(* IEC 61131-3 sources: Mizera_Tube/Plc (part 3) *)

(* ---- LASER.plc ---- *)
*******************************************************************************
*   LASER.PLC
*   ESAutomotion
*   LASER machine
*******************************************************************************
#funcdec "FLP.plc"
#funcdec "RestFB.plc"
VAR
#include "Cnc.inc"

#include "RemContr.inc"

HoerbEnabCond: BOOL; * Hoerbiger prop. valve enable conditions
TOF_HBPROP: TOF;
#defcom TOF_HBPROP.Q Hoerbiger prop valve enable delayed

appoggio:             BOOL;

TP_HOLD_Tip:                TP;
TP_HOLD_Noz:                TP;

F_DIS_MANAPA:               F_TRIG;

R_TRIG_PRGRUN:              R_TRIG; * Fronte salita start programma
R_TRIG_PRGRUN2:             R_TRIG; * Fronte salita start programma
F_TRIG_PRGRUN:              F_TRIG; * Fronte discesa start programma

R_TRIG0:                    R_TRIG;
TON_ST:                        TON;

*manual cut
TP_EXE_REQ:                 TP;
FTRIG_PRUN:                 F_TRIG;
TP_EXE_REQ2:                TP;
FTRIG_PRUN2:                F_TRIG;
RTRIG_Xstart:               R_TRIG;
RTRIG_Xend:                 R_TRIG;
RTRIG_Ystart:               R_TRIG;
RTRIG_Yend:                 R_TRIG;
RTRIG_REQ_BREAK:            R_TRIG;
*
* microjoint alg
firScan:                   DWORD;                * Initialization of filter
RTRIG_FIR_INIT:           R_TRIG;
error:                     DWORD;
TON_VALID_DATA:              TON;

TON_DISABLE_BEAM:            TON;
RTRIG_CAL_FILTER:         R_TRIG;
velMaxAlg:                 DWORD;                 * set point speed to have filter at 0
RTRIG_START_LEAD:         R_TRIG;
FTRIG_START_LEAD:         F_TRIG;
posXinitlead:              DWORD;
posYinitlead:              DWORD;
posXendlead:               DWORD;
posYendlead:               DWORD;
PosIntInitLead:            DWORD;
PosIntendLead:             DWORD;
microJoinfactor:           DWORD;        * need to comensate the possible radius during lead in
percReduction:             DWORD;
LinearDistance:            DWORD;
RealLeadDistance:          DWORD;
distX:                     DWORD;
distY:                     DWORD;
indexLeadIn:               DWORD;        * if  indexLeadIn = 314 lead in is a semicircumference
Ftrig_LeadTest:           F_TRIG;

RTRIG_COUNT_PIERC:        R_TRIG;
rtrig_ResPiercCounter:    R_TRIG;
rtrig_ResPiercCounter_2:  R_TRIG;
MicroJointime:         DWORD;

* wrong operation protection

RTRIG_NOPIERC:            R_TRIG;
RTRIG_ALLPIERC:           R_TRIG;
RTRIG_NOLEAD:             R_TRIG;
RTRIG_RES_GEOM:           R_TRIG;
RTRIG_RES_PIECE:          R_TRIG;
FTRIG_RES_AUTO_CLEAN:     F_TRIG;
RTRIG_WORK_ENAB:          R_TRIG;

TP_BUZZER:              TP;         * Buzzer timer
TP_HOLD_BODY:           TP;

TON_REMOVE_ALARM:       TON;
RTRIG_ORIG19:           R_TRIG;
RTRIG_BLOCK_S:          R_TRIG;

RTRIG_MANSEL_P:         R_TRIG;         * Selettore manuale (potenza/duty/frequenza)
RTRIG_MANSEL_M:         R_TRIG;         * Selettore manuale (potenza/duty/frequenza)

Restart:                Restart_Cut;

END_VAR

VAR_IN_OUT
#include "mem.inc"
END_VAR

#include "Iol.inc"

******************************************************************************
* FUNCTION LASER_IN
******************************************************************************
FUNCTION LASER_IN

**@@@ INP_TEST    * Digital Inputs test management

******************************************************************************
*   Gestione selettore manuale x cambiamento valori potenza/duty/frequenza
******************************************************************************
CAL  RTRIG_MANSEL_P (CLK:=%SoftBtn1.0)
CAL  RTRIG_MANSEL_M (CLK:=%SoftBtn1.1)

*** INC

LD   ON_ONE_SCAN                   ** PLCFLAGS.8  Flag on alla prima scansione PLC
OR (
LD   ManSelector            *(rgGui6)Selettore manuale potenza/duty/frequenza
LE   0
)
OR (
LD   ManSelector            *(rgGui6)Selettore manuale potenza/duty/frequenza
GT   3
)
JMPCN man_sel_init

LD   100
ST   ManSelectorPOW         *(rgGui7)Selettore manuale POTENZA: ultimo valore impostato
ST   ManSelectorDUTY        *(rgGui8)Selettore manuale DUTY: ultimo valore impostato
ST   ManSelectorFREQ        *(rgGui9)Selettore manuale FREQUENCY: ultimo valore impostato

man_sel_init:

LD   RTRIG_MANSEL_P.Q
AND (
LD   ManSelector            *(rgGui6)Selettore manuale potenza/duty/frequenza
EQ   1
)
JMPCN no_pow_inc

LD   ManSelectorPOW         *(rgGui7)Selettore manuale POTENZA: ultimo valore impostato
ADD  1
ST   ManSelectorPOW         *(rgGui7)Selettore manuale POTENZA: ultimo valore impostato

no_pow_inc:
LD   RTRIG_MANSEL_P.Q
AND (
LD   ManSelector            *(rgGui6)Selettore manuale potenza/duty/frequenza
EQ   2
)
JMPCN no_duty_inc

LD   ManSelectorDUTY        *(rgGui8)Selettore manuale DUTY: ultimo valore impostato
ADD  5
ST   ManSelectorDUTY        *(rgGui8)Selettore manuale DUTY: ultimo valore impostato

no_duty_inc:
LD   RTRIG_MANSEL_P.Q
AND (
LD   ManSelector            *(rgGui6)Selettore manuale potenza/duty/frequenza
EQ   3
)
JMPCN no_freq_inc

LD   ManSelectorFREQ        *(rgGui9)Selettore manuale FREQUENCY: ultimo valore impostato
ADD  5
ST   ManSelectorFREQ        *(rgGui9)Selettore manuale FREQUENCY: ultimo valore impostato

no_freq_inc:

*** DEC

LD   RTRIG_MANSEL_M.Q
AND (
LD   ManSelector            *(rgGui6)Selettore manuale potenza/duty/frequenza
EQ   1
)
JMPCN no_pow_dec

LD   ManSelectorPOW         *(rgGui7)Selettore manuale POTENZA: ultimo valore impostato
SUB  1
ST   ManSelectorPOW         *(rgGui7)Selettore manuale POTENZA: ultimo valore impostato

no_pow_dec:
LD   RTRIG_MANSEL_M.Q
AND (
LD   ManSelector            *(rgGui6)Selettore manuale potenza/duty/frequenza
EQ   2
)
JMPCN no_duty_dec

LD   ManSelectorDUTY        *(rgGui8)Selettore manuale DUTY: ultimo valore impostato
SUB  5
ST   ManSelectorDUTY        *(rgGui8)Selettore manuale DUTY: ultimo valore impostato

no_duty_dec:
LD   RTRIG_MANSEL_M.Q
AND (
LD   ManSelector            *(rgGui6)Selettore manuale potenza/duty/frequenza
EQ   3
)
JMPCN no_freq_dec

LD   ManSelectorFREQ        *(rgGui9)Selettore manuale FREQUENCY: ultimo valore impostato
SUB  5
ST   ManSelectorFREQ        *(rgGui9)Selettore manuale FREQUENCY: ultimo valore impostato

no_freq_dec:

*** CONTROLLO VALORE MINIMO/MASSIMO

LD   ManSelectorPOW         *(rgGui7)Selettore manuale POTENZA: ultimo valore impostato
LT   0
JMPCN no_pow_zero
LD   0
ST   ManSelectorPOW         *(rgGui7)Selettore manuale POTENZA: ultimo valore impostato
no_pow_zero:
LD   ManSelectorPOW         *(rgGui7)Selettore manuale POTENZA: ultimo valore impostato
GT   120
JMPCN no_pow_max
LD   120
ST   ManSelectorPOW         *(rgGui7)Selettore manuale POTENZA: ultimo valore impostato
no_pow_max:

LD   ManSelectorDUTY        *(rgGui8)Selettore manuale DUTY: ultimo valore impostato
LT   0
JMPCN no_duty_zero
LD   0
ST   ManSelectorDUTY        *(rgGui8)Selettore manuale DUTY: ultimo valore impostato
no_duty_zero:
LD   ManSelectorDUTY        *(rgGui8)Selettore manuale DUTY: ultimo valore impostato
GT   120
JMPCN no_duty_max
LD   120
ST   ManSelectorDUTY        *(rgGui8)Selettore manuale DUTY: ultimo valore impostato
no_duty_max:

LD   ManSelectorFREQ        *(rgGui9)Selettore manuale FREQUENCY: ultimo valore impostato
LT   0
JMPCN no_freq_zero
LD   0
ST   ManSelectorFREQ        *(rgGui9)Selettore manuale FREQUENCY: ultimo valore impostato
no_freq_zero:
LD   ManSelectorFREQ        *(rgGui9)Selettore manuale FREQUENCY: ultimo valore impostato
GT   120
JMPCN no_freq_max
LD   120
ST   ManSelectorFREQ        *(rgGui9)Selettore manuale FREQUENCY: ultimo valore impostato
no_freq_max:

*** VALORI DI USCITA PER LsrGest.plc

LD   0
ST   ManSelectorPOW_out         *(gPlc30)Selettore manuale POTENZA: ultimo valore impostato (valore di uscita per LsrGest)
ST   ManSelectorDUTY_out        *(gPlc30)Selettore manuale DUTY: ultimo valore impostato (valore di uscita per LsrGest)
ST   ManSelectorFREQ_out        *(gPlc30)Selettore manuale FREQUENCY: ultimo valore impostato (valore di uscita per LsrGest)

LD   ManSelector            *(rgGui6)Selettore manuale potenza/duty/frequenza
EQ   1
JMPCN no_pow

LD   100
ST   ManSelectorDUTY        *(rgGui8)Selettore manuale DUTY: ultimo valore impostato
ST   ManSelectorFREQ        *(rgGui9)Selettore manuale FREQUENCY: ultimo valore impostato
JMP  no_freq

no_pow:
LD   ManSelector            *(rgGui6)Selettore manuale potenza/duty/frequenza
EQ   2
JMPCN no_duty

LD   100
ST   ManSelectorPOW         *(rgGui7)Selettore manuale POTENZA: ultimo valore impostato
ST   ManSelectorFREQ        *(rgGui9)Selettore manuale FREQUENCY: ultimo valore impostato
JMP  no_freq

no_duty:
LD   ManSelector            *(rgGui6)Selettore manuale potenza/duty/frequenza
EQ   3
JMPCN no_freq

LD   100
ST   ManSelectorPOW         *(rgGui7)Selettore manuale POTENZA: ultimo valore impostato
ST   ManSelectorDUTY        *(rgGui8)Selettore manuale DUTY: ultimo valore impostato

LD   %TabLsr0.L_CutFreq
MUL (
LD   ManSelectorFREQ        *(rgGui9)Selettore manuale FREQUENCY: ultimo valore impostato
SUB  100                    * 100%
)
DIV  100                    * 100 %
ST   ManSelectorFREQ_out        *(gPlc30)Selettore manuale FREQUENCY: ultimo valore impostato (valore di uscita per LsrGest)

no_freq:

******************************************************************************
*   Copia il valore della potenza massima sulla variabile usata dalla GUI
******************************************************************************
LD   %LsrGest0.ParMaxPower
ST   PotenzaMaxLaser            **(rLsGui17)Potenza massima Laser

******************************************************************************
* Safety for axes when operator move in jog the axes
CAL  TON_REMOVE_ALARM (IN:=%PLCerr7.21,PT:=5000)    * Axes cannot move, not safe movement

LD   OrderMoveYPosit               ** (LsPlc26.5) Order of movement positive dir for Y
OR   OrderMoveYNegat               ** (LsPlc26.6) Order of movement negative dir for Y
OR   OrderMoveXPosit               ** (LsPlc26.3) Order of movement positive dir for X
OR   OrderMoveXNegat               ** (LsPlc26.4) Order of movement negative dir for X
OR   Pul_Reset                     ** (gPlc0.3)Reset pushbutton
OR   TON_REMOVE_ALARM.Q        * Reset of the alarm
OR   PRGRUN_CN0                    ** M0.0 cn0.rc8.0  Programma in corso
R    %PLCerr7.21               * Axes cannot move, not safe movement

LD   %CalPipe0.General0.5       * pipe is along Y axis
AND  %cn3.cc1.5                 * W axis configured
ANDN PRGRUN_CN0                    ** M0.0 cn0.rc8.0  Programma in corso
ANDN BCI_TAR                       ** rc0.8  Selettore modi operativi su REF (taratura)
JMPCN noPipeY

  * hold moving if the bridge in in the middle of the machine and
  * the operator move X in pipe side
  LD   %ax28.ra4                  * y axis position
  SUB  3000
  GT   %tab1.t_ttab.t_oart.t_dY   * pipe offset along y axis
  OR  (
  LD   %ax29.ra4
  LE  (
  LD   %ax29.pa22
  SUB  10000
  )
  )
  AND  (
  LD   %ax27.ra4                  * x axis position
  LE   (
  LD   %ax27.pa21
  ADD  SafePipeZone                  ** (%LSRCostK9) Safety distance from axis limit in pipe management
   )
  )
  AND  (
  LD  %tab1.t_ttab.t_oart.t_dX
  LT  0
  )
  AND OrderMoveXNegat                ** (LsPlc26.4) Order of movement negative dir for X
 ***************************
  OR  ( * x is in the pipe side but head is not up
  LD   %ax27.ra4                  * x axis position
  LT   (
  LD   %ax27.pa21
  ADD  SafePipeZone                  ** (%LSRCostK9) Safety distance from axis limit in pipe management
   )
  AND (
  LD   %ax29.ra4
  LE  (
  LD   %ax29.pa22
  SUB  10000
    )
   )
  AND  OrderMoveXPosit               ** (LsPlc26.3) Order of movement positive dir for X
  ANDN (
  LD   %ax28.ra4                  * y axis position
  SUB  3000
  GT   %tab1.t_ttab.t_oart.t_dY   * pipe offset along y axis
  )
  AND  (
  LD  %tab1.t_ttab.t_oart.t_dX
  LT  0
  )
  )
 **************************
  OR  (  * same condition, in case the pipe is in positive direction of X axis
   LD   %ax28.ra4                  * y axis position
   SUB  3000
   GT   %tab1.t_ttab.t_oart.t_dY   * pipe offset along y axis
   OR  (
   LD   %ax29.ra4
   LE  (
   LD   %ax29.pa22
   SUB  10000
    )
   )
   AND  (
   LD   %ax27.ra4                  * x axis position
   GE   (
   LD   %ax27.pa22
   SUB  SafePipeZone                  ** (%LSRCostK9) Safety distance from axis limit in pipe management
    )
   )
   AND  (
   LD  %tab1.t_ttab.t_oart.t_dX
   GT  0
   )
   AND  OrderMoveXPosit               ** (LsPlc26.3) Order of movement positive dir for X
  )
 ***************************
  OR  ( * x is in the pipe side but head is not up
  LD   %ax27.ra4                  * x axis position
  GE   (
  LD   %ax27.pa22
  SUB  SafePipeZone                  ** (%LSRCostK9) Safety distance from axis limit in pipe management
   )
  AND (
  LD   %ax29.ra4
  LE  (
  LD   %ax29.pa22
  SUB  10000
    )
   )
  AND  OrderMoveXNegat               ** (LsPlc26.4) Order of movement negative dir for X
  ANDN (
  LD   %ax28.ra4                  * y axis position
  SUB  3000
  GT   %tab1.t_ttab.t_oart.t_dY   * pipe offset along y axis
  )
  AND  (
  LD  %tab1.t_ttab.t_oart.t_dX
  GT  0
   )
  )
 **************************
  ST  HoldSafePipeX                  ** (LsPlc26.2) Hold moving for X axis, not allow manual movement in pipe area

  LD   %ax27.ra4                  * x axis position
  LT   (
  LD   %ax27.pa21
  ADD  SafePipeZone                  ** (%LSRCostK9) Safety distance from axis limit in pipe management
   )
  AND  (
  LD  %tab1.t_ttab.t_oart.t_dX
  LT  0
  )
  AND (
  LD  OrderMoveYPosit                ** (LsPlc26.5) Order of movement positive dir for Y
  OR  OrderMoveYNegat                ** (LsPlc26.6) Order of movement negative dir for Y
  )
  OR  (
   LD   %ax27.ra4                 * x axis position
   GT   (
   LD   %ax27.pa22
   SUB  SafePipeZone                  ** (%LSRCostK9) Safety distance from axis limit in pipe management
    )
    AND  (
    LD  %tab1.t_ttab.t_oart.t_dX
    GT  0
   )
    AND (
    LD  OrderMoveYPosit                ** (LsPlc26.5) Order of movement positive dir for Y
    OR  OrderMoveYNegat                ** (LsPlc26.6) Order of movement negative dir for Y
   )
  )
  ST   HoldSafePipeY                 ** (LsPlc26.7) Hold moving for Y axis, not allow manual movement in pipe area

noPipeY:

* Safety for axes when operator move in jog the axes
* NEED TO BE TESTED,ACTUALLY MACHINE HAVE PIPE ALONG y

LD   %CalPipe0.General0.4       * pipe is along X axis
AND  %cn3.cc1.5                 * W axis configured
ANDN PRGRUN_CN0                    ** M0.0 cn0.rc8.0  Programma in corso
ANDN BCI_TAR                       ** rc0.8  Selettore modi operativi su REF (taratura)
JMPCN noPipeX

  LD   %ax27.ra4                  * x axis position
  SUB  3000
  GT   %tab1.t_ttab.t_oart.t_dX   * pipe offset along x axis
  AND  (
  LD   %ax28.ra4                  * y axis position
  LT   (
  LD   %ax28.pa21
  ADD  SafePipeZone                  ** (%LSRCostK9) Safety distance from axis limit in pipe management
   )
  )
  AND  (
  LD  %tab1.t_ttab.t_oart.t_dY
  LT  0
  )
  AND OrderMoveYNegat                ** (LsPlc26.6) Order of movement negative dir for Y
  OR  (
   LD   %ax27.ra4                  * x axis position
   SUB  3000
   GT   %tab1.t_ttab.t_oart.t_dX   * pipe offset along y axis
   AND  (
   LD   %ax28.ra4                  * y axis position
   GT   (
   LD   %ax28.pa22
   SUB  SafePipeZone                  ** (%LSRCostK9) Safety distance from axis limit in pipe management
    )
   )
   AND  (
   LD  %tab1.t_ttab.t_oart.t_dY
   GT  0
   )
   AND  OrderMoveYPosit               ** (LsPlc26.5) Order of movement positive dir for Y
  )
  ST  HoldSafePipeY                  ** (LsPlc26.7) Hold moving for Y axis, not allow manual movement in pipe area

  LD   %ax28.ra4                   * y axis position
  LT   (
  LD   %ax28.pa21
  ADD  SafePipeZone                  ** (%LSRCostK9) Safety distance from axis limit in pipe management
   )
  AND  (
  LD  %tab1.t_ttab.t_oart.t_dY
  LT  0
  )
  AND (
  LD  OrderMoveYPosit                ** (LsPlc26.5) Order of movement positive dir for Y
  OR  OrderMoveYNegat                ** (LsPlc26.6) Order of movement negative dir for Y
  )
  OR  (
   LD   %ax28.ra4                  * y axis position
   GT   (
   LD   %ax28.pa22
   SUB  SafePipeZone                  ** (%LSRCostK9) Safety distance from axis limit in pipe management
    )
    AND  (
    LD  %tab1.t_ttab.t_oart.t_dY
    GT  0
   )
    AND (
    LD  OrderMoveYPosit                ** (LsPlc26.5) Order of movement positive dir for Y
    OR  OrderMoveYNegat                ** (LsPlc26.6) Order of movement negative dir for Y
   )
  )
  ST   HoldSafePipeX                 ** (LsPlc26.2) Hold moving for X axis, not allow manual movement in pipe area

noPipeX:

LD   HoldSafePipeX                 ** (LsPlc26.2) Hold moving for X axis, not allow manual movement in pipe area
OR   HoldSafePipeY                 ** (LsPlc26.7) Hold moving for Y axis, not allow manual movement in pipe area
S    %PLCerr7.21                    * Axes cannot move, not safe movement

******************************************************************************
******************************************************************************
*   BUZZER MANAGEMENT
******************************************************************************
LD   PRGRUN_CN0                    ** M0.0 cn0.rc8.0  Programma in corso
ST   appoggio

CAL  TP_BUZZER(IN=PRGRUN_CN0,PT=%Cost_User20) ** Buzzer timer

LD   TP_BUZZER.Q
ST	 O_O_BUZZER_START_CIC           ** Star cycle buzzer

******************************************************************************
CAL  TP_HOLD_Tip(IN=%PLCerr5.4,PT=500) **PLC Err 164 Tip touch (A11=1, A14=0, A15=0 in normal operation)
CAL  TP_HOLD_Noz(IN=%PLCerr5.6,PT=1000) **PLC Err 166 Nozzle lost (A11=1, A14=0, A15=1 in normal operation)
CAL  TP_HOLD_BODY (IN:=%PLCerr5.5,PT:=1000)                    **PLC Err 165 Body touch (A11=1, A14=1, A15=0 in normal operation)

LD   TP_HOLD_Tip.Q
OR   TP_HOLD_Noz.Q
OR   TP_HOLD_BODY.Q
ST   StopUsrPlc                    ** (gPlc2.22)Richiesta STOP da User_Plc

**************************************
*& Set TAB value for startup (retentive)
**
LD      ON_ONE_SCAN                ** PLCFLAGS.8  Flag on alla prima scansione PLC
JMPCN   No_FirstScan
  LD      guiTAB_Sinottico           ** (rGui10)GUI TAB Sinottico for Quotes
  EQ      0
  JMPCN   No_TabEqZero
    LD      1
    ST      guiTAB_Sinottico           ** (rGui10)GUI TAB Sinottico for Quotes
No_TabEqZero:
No_FirstScan:

CAL R_TRIG0(CLK=%PLCFLAGS.10)

LD   R_TRIG0.Q
JMPCN CNT_MP

LD   Timesec                       ** (R123) Tempo secondi
ADD  1
ST   Timesec                       ** (R123) Tempo secondi

CNT_MP:

LD   Timesec                       ** (R123) Tempo secondi
DIV  3600
ST   TimeOur                       ** (R124) Tempo ore
****************************************************************

****************************************************************
* Tempo Taglio In Corso
****************************************************************

CAL  TON_ST(IN:=StartTimer,PT:=1000) ** Start tim

LD   %cn0.rc8.0                    * Programma in corso cn0
AND  TON_ST.Q                     * Start tim
ANDN PRGSTOP_CN0                   ** (cn0.rc8.1)  Programma interrotto CN0
AND  R_TRIG0.Q                     * Impulso incremento secondi
JMPCN TIMECUT

* Contasecondi

LD   TimeSecProg                   ** (R125) Conteggio Secondi Tempo Programma Taglio in corso
ADD  1
ST   TimeSecProg                   ** (R125) Conteggio Secondi Tempo Programma Taglio in corso

TIMECUT:

CAL R_TRIG_PRGRUN(CLK=%cn0.rc8.0)	 ** Fronte salita start programma

LD   R_TRIG_PRGRUN.Q
JMPCN ResCount

LD   0
ST   TimeSecProg                   ** (R125) Conteggio Secondi Tempo Programma Taglio in corso
ST   TimeMinProg                   ** (R126) Conteggio Minuti Tempo Programma Taglio in corso

ResCount:

LD   Pul_Reset                     ** (gPlc0.3)Reset pushbutton
JMPCN no_zero
LD   0
ST   StartTimer                    ** Start tim
no_zero:

*******************************************************************************
*   Restart Taglio
*******************************************************************************
LD   PRGRUN_CN0
ST   Restart.xProg_Run

LD   %PLCerr5.4                    **PLC Err 164 Tip touch (A11=1, A14=0, A15=0 in normal operation)
AND  EnTiptouchRetrace
AND  BevelHeadSyncG800              * Traccia in esecuzione
ST   Restart.xTip_Touch

LD   VRTCIncSetPReached
ST   Restart.xZupExecuted

LD   PRGSTOP_CN0
ST   Restart.xMachineInHold

LD   %LSRCostK13                    ** (LSRCostK13) Numero tentativi per tip touch con gestione autorestart
ST   Restart.xAttempts

LD   RetraceCommBack
ST   Restart.xRetraceOn

CAL  Restart

LD   Restart.yStartProg
ST   StartAftTipTouch              ** (LsPlc47.2) Start after tip touch

LD   Restart.yStartRetrace
ST   JogCommandTipTouch            ** (LsPlc47.0) Automatic jog command for tip touch

LD   Restart.yZupRequest
ST   EnPosiz                       * (LsPlc47.3) Abilitaz. posiz. Asse Z

LD   Restart.yInibTipTouch
AND  EnTiptouchRetrace
ST   InibTipTouchAllarm            ** M100.22 Inibizione allarme Tip Touch per restart ciclo

**********************************************************************************
* enable/disable automatic height control manual cut

LD   %cn0.rc9            * Channel 0 M-Functions register
EQ   4001
AND  %cn0.rc8.4          * Channel 0 M-Functions Strobe
S    M4001_REQ           * (LsPlc47.14) M4001 request to enable height threshold detection

LD   %cn0.rc9            * Channel 0 M-Functions register
EQ   4002
AND  %cn0.rc8.4          * Channel 0 M-Functions Strobe
ORN  PRGRUN_CN0                    ** M0.0 cn0.rc8.0  Programma in corso
R    M4001_REQ           * (LsPlc47.14) M4001 request to enable height threshold detection

*
********************************************************************************
* Turn off laser by distance to go

LD   EnMicroJoint                  ** (%rLsGui29.4) Enable microjoint option
JMPCN no_microjoint_func

* Compensation if the lead in is not straight

CAL  RTRIG_START_LEAD (CLK:=LeadInStart) ** SignaL lead in in progress

LD   RTRIG_START_LEAD.Q
JMPCN acuXYdist

LD   %ax27.ra4
ST   posXinitlead

LD   %ax28.ra4
ST   posYinitlead

LD   %ax21.ra25
ST   PosIntInitLead

acuXYdist:

CAL  FTRIG_START_LEAD (CLK:=LeadInStart) ** SignaL lead in in progress

LD   FTRIG_START_LEAD.Q
JMPCN endLead

LD   %ax27.ra4
ST   posXendlead

LD   %ax28.ra4
ST   posYendlead

LD   %ax21.ra25
ST   PosIntendLead

LD   PosIntendLead
SUB  PosIntInitLead
ST   RealLeadDistance

* Calc linear distance

LD   posXendlead
SUB  posXinitlead
ST   distX

LD   posYendlead
SUB  posYinitlead
ST   distY

LD   0
HYPOT (X=distX,Y=distY)
ST   LinearDistance

LD   0
ST   microJoinfactor               ** need to comensate the possible radius during lead in

LD   RealLeadDistance
GT   LinearDistance
JMPCN changecompens

LD   RealLeadDistance
MUL  2
MUL  100
DIV  LinearDistance
ST   indexLeadIn                   ** if  indexLeadIn = 314 lead in is a semicircumference

*y=mx+c => x=indexLeadIn  Y=0-100% X=200-314
LD   indexLeadIn                   ** if  indexLeadIn = 314 lead in is a semicircumference
MUL  87719
DIV  1000
SUB  17544
DIV  100
ST   percReduction

*LD   indexLeadIn                       * if  indexLeadIn = 314 lead in is a semicircumference
*MUL  100
*DIV  314
*ST   percReduction

LD   percReduction
GT   100
JMPCN limitperc

LD   100
ST   percReduction

limitperc:

LD   SpaceForLeadCom               ** (%LsGui82) Costant to compensate no linear lead in (max value of compensation)
MUL  percReduction
DIV  100
ST   microJoinfactor               ** need to comensate the possible radius during lead in
changecompens:

endLead:

*LD   InterpolatResidual
LD   %ax21.ra29
LT   (
LD   MicroJointDist                ** (rLsGui25) Distance for microjoint
ADD  microJoinfactor               ** need to comensate the possible radius during lead in
)
AND  %ax21.ra8.21
ST   appoggio

* Interpolation of filter time to compensate the output delay
****

LD   666667                             * 40000 mm/min
MUL  -1
ST   velMaxAlg                     ** set point speed to have filter at 0

CAL  RTRIG_CAL_FILTER (CLK:=appoggio)

LD   RTRIG_CAL_FILTER.Q
JMPCN nofilCal
LD   FilterForMicroJ               ** (rLsGui26) Microjoint FIR time (NOT USED)
MUL  (
LD   %ax21.ra28                       * interpolator speed (micro/sec) Proc.Principale CN0
ADD  velMaxAlg                     ** set point speed to have filter at 0
)
DIV  velMaxAlg                     ** set point speed to have filter at 0
ST   MicroJointime

nofilCal:

CAL  TON_DISABLE_BEAM (IN:=appoggio,PT:=MicroJointime) * Data valid for microjoint

LD   TON_DISABLE_BEAM.Q
ANDN (
LD   %LsIso11
EQ   4
OR   (
LD   %LsIso11
EQ   5
)
OR   INP_flyCutModeON                 ** application turn flyCut mode ON
)
S    TurnOffLaser                  ** (LsPlc47.19) Turn off laser from microjoint algorithm

LD   enabcopy                      ** test copia
JMPC nocopy

LD   %PlPlc21
ST   %PlPlc22           * 3

LD   %PlPlc20
ST   %PlPlc21           * 2

LD   %ax21.ra29
ST   %PlPlc20           * 1

nocopy:

LD   TurnOffLaser                  ** (LsPlc47.19) Turn off laser from microjoint algorithm
S    enabcopy                      ** test copia

****

LD   piercing_run                  ** (LsPlc37) Piercing in run
***ORN  %ax21.ra8.21                     * Data valid for microjoint  VA VIA TROPPO PRESTO
ORN  PRGRUN_CN0                    ** M0.0 cn0.rc8.0  Programma in corso
R    TurnOffLaser                  ** (LsPlc47.19) Turn off laser from microjoint algorithm

CAL  Ftrig_LeadTest (CLK:=PRGRUN_CN0) ** M0.0 cn0.rc8.0  Programma in corso

LD   Ftrig_LeadTest.Q
OR   Pul_Reset                     ** (gPlc0.3)Reset pushbutton
JMPCN no_res_var
LD   0
ST   LeadInStart                   ** SignaL lead in in progress
no_res_var:
no_microjoint_func:
******************************************************************************************
END_FUNCTION

******************************************************************************
******************************************************************************
******************************************************************************
* FUNCTION LASER_M
******************************************************************************
******************************************************************************
******************************************************************************
FUNCTION LASER_M

LD   ALWAYS_ZERO                   ** PLCFLAGS.0  Flag sempre stato off
ST   PresetDaErrore                ** (gPlc2.2)Rich. Preset/Allineamento quota slave a master per errore allin.

LD   ALWAYS_ZERO                   ** PLCFLAGS.0  Flag sempre stato off
ST   Stop_Req_PLC                  ** (gPlc0.12)Richiesta stop ciclo da PLC.plc

LD   ALWAYS_ZERO                   ** PLCFLAGS.0  Flag sempre stato off
ST   Blav_Req_PLC                  ** (gPlc0.13)Richiesta blocco avanzamento XY da PLC.plc

***
Gest_Assi
***
Macch_Reset
***
Barriere
***
Pneumatico
***
GestGas
GasProp
***
REMOTE_DISPLAY
***
LOG
***
CLAMP_SUPPORT
***
PIPE_CALIBRATION
***
LuciMacc
***

END_FUNCTION

******************************************************************************
******************************************************************************
******************************************************************************
* FUNCTION LASER_OUT
******************************************************************************
******************************************************************************
******************************************************************************
FUNCTION LASER_OUT

CAL  R_TRIG_PRGRUN2(CLK=%cn0.rc8.0)
CAL  F_TRIG_PRGRUN(CLK=%cn0.rc8.0)

******************************************************************************
*   WELDING management
******************************************************************************
LD   %LSRPlcOp0.22                 ** Pipe Welding function enabling
JMPCN NoWeldingM

LD   R_TRIG_PRGRUN2.Q
OR   F_TRIG_PRGRUN.Q
OR (
LD   Pul_Reset                     ** (gPlc0.3)Reset pushbutton
ANDN PRGRUN_CN0                    ** M0.0 cn0.rc8.0  Programma in corso
)
R    WeldingSensorPiston

LD   WeldingSensorPiston
ST   O_O_WELDING_PISTON

NoWeldingM:

******************************************************************************
*   Aspirator
******************************************************************************
Aspiraz

******************************************************************************
*   Hoerbiger proportional valve
******************************************************************************
LD   O_O_EV_OPEN_N2                ** Elettrovalvola apertura Azoto
AND  GasPVHoerbiger                ** M107.22 Cutting gas prop. valve type hoerbiger
ST   O_O_EV_OPEN_N2_HOERB          ** Hoerbiger: N2 ev

LD   O_O_EV_OPEN_O2                ** Elettrovalvola apertura Ossigeno
AND  GasPVHoerbiger                ** M107.22 Cutting gas prop. valve type hoerbiger
ST   O_O_EV_OPEN_O2_HOERB          ** Hoerbiger: O2 ev

LD   O_O_EV_OPEN_ARIA              ** Elettrovalvola apertura Aria taglio
AND  GasPVHoerbiger                ** M107.22 Cutting gas prop. valve type hoerbiger
ST   O_O_EV_OPEN_ARIA_HOERB        ** Hoerbiger: air ev

***************************************
* Enable valve for oxygen and nitrogen
***************************************
LD   %config_machine29             ** Proportional valve manage only with OXYGEN
EQ   0
AND  O_O_EV_OPEN_N2                ** Elettrovalvola apertura Azoto
OR   O_O_EV_OPEN_O2                ** Elettrovalvola apertura Ossigeno
ST   HoerbEnabCond                 ** Hoerbiger prop. valve enable conditions

CAL  TOF_HBPROP(IN:=HoerbEnabCond,PT:=60000) ** Hoerbiger prop. valve enable conditions

LD   TOF_HBPROP.Q                  ** Hoerbiger prop valve enable delayed
ST   O_O_ENAB_VALVE_HOERB          ** Enable proportional valve for oxygen (Hoerbiger)

*PILOTAGGIO HOERBIGER
LD   O_O_EV_OR_ALLGAS              ** M90.15 Elettrovalvola apertura di almeno un gas
AND  GasPVHoerbiger                ** M107.22 Cutting gas prop. valve type hoerbiger
OR   O_O_CALIB_REQ_HOERB           ** Hoerbiger: calibration request
ST   O_O_PILOT_HOERB               ** Hoerbiger: gas command ev

**********************************************************************

**********************************************************************
*******************************************************************************
* Manual Cut Request
*******************************************************************************

LD    guiManualReq                 ** (gGui22.1) Manual cut request
AND   %cn0.rgc0.3                     * rgc0.3 Canale in JOG o INC
ST    appoggio

CAL  TP_EXE_REQ(IN:=appoggio,PT:=300)

LD   TP_EXE_REQ.Q
S    exeaux_for_mancut               ** (LsPlc47.8) manual cut request

CAL  FTRIG_PRUN (CLK:=%cn0.rc8.0)

LD   Pul_Reset                     ** (gPlc0.3)Reset pushbutton
OR   FTRIG_PRUN.Q
OR   I_I_EMERGENZA                 ** Machine OK (no EMERG.)
OR   EMER_GEN                      ** M0.10 Emergenza generale
R    exeaux_for_mancut               ** (LsPlc47.8) manual cut request

CAL  RTRIG_Xstart (CLK:=guiAcqXstart) ** (gGui22.2) Manual cut: acquire X start quota
CAL  RTRIG_Xend (CLK:=guiAcqXend)  ** (gGui22.3) Manual cut: acquire X end quota
CAL  RTRIG_Ystart (CLK:=guiAcqYstart) ** (gGui22.4) Manual cut: acquire Y start quota
CAL  RTRIG_Yend (CLK:=guiAcqYend)  ** (gGui22.5) Manual cut: acquire Y end quota

LD   RTRIG_Xstart.Q
ANDN %cn0.rc8.0
JMPCN NoAcq1

LD   %ax27.ra4
ST   qCut_X_start                  ** (rLsGui48) Manual cut: X quota start

NoAcq1:
LD   RTRIG_Xend.Q
ANDN %cn0.rc8.0
JMPCN NoAcq2

LD   %ax27.ra4
ST   qCut_X_end                    ** (rLsGui49) Manual cut: X quota end

NoAcq2:
LD   RTRIG_Ystart.Q
ANDN %cn0.rc8.0
JMPCN NoAcq1_

LD   %ax28.ra4
ST   qCut_Y_start                  ** (rLsGui50) Manual cut: Y quota start

NoAcq1_:
LD   RTRIG_Yend.Q
ANDN %cn0.rc8.0
JMPCN NoAcq2_

LD   %ax28.ra4
ST   qCut_Y_end                    ** (rLsGui51) Manual cut: Y quota end

NoAcq2_:
**********************************************************************
* Break Point positioning

CAL  RTRIG_REQ_BREAK (CLK:=RemContrBreakPoint) ** Xhc_Puls.7  Break point positioning request*

LD   RTRIG_REQ_BREAK.Q
S    BreakPosReq               ** (LsPlc47.17) Request break point positioning

LD   Pul_Reset                     ** (gPlc0.3)Reset pushbutton
OR   FTRIG_PRUN.Q
OR   I_I_EMERGENZA                 ** Machine OK (no EMERG.)
OR   EMER_GEN                      ** M0.10 Emergenza generale
R    BreakPosReq               ** (LsPlc47.17) Request break point positioning

**********************************************************************

**********************************************************************
* Piercing counter

CAL  RTRIG_COUNT_PIERC (CLK:=PiercingInRun.0)   * (LsPlc70) Piercing in run

LD   RTRIG_COUNT_PIERC.Q            * (LsPlc70) Piercing in run
ANDN %PlcOp0.2                     ** DryRun
ANDN (                              * customer line for marking
LD   CurrentLineExecute            ** (LsIso11) Current cutting line parameter to execute
EQ   4
)
ANDN (                              * customer line for film burning
LD   CurrentLineExecute            ** (LsIso11) Current cutting line parameter to execute
EQ   5
)
ANDN INP_flyCutModeON              ** application turn flyCut mode ON
JMPCN no_pierc_count

LD   PiercCounter                  ** (%C71) Piercing counter
ADD  1
ST   PiercCounter                  ** (%C71) Piercing counter

no_pierc_count:

CAL rtrig_ResPiercCounter_2 (CLK:=AutoNozzleClean) ** (%rLsGui29.9) Nozzle clean active

LD   BtnResetCounter               ** (LsGui32.28) Reset counter of piercing
OR   rtrig_ResPiercCounter_2.Q
OR   Nozzle_clean_run               * (C26.1) Nozzle cleaning in run
ST   appoggio

CAL  rtrig_ResPiercCounter (CLK:=appoggio) *  Reset counter of piercing

LD   rtrig_ResPiercCounter.Q
JMPCN  norescounter

LD   0
ST   PiercCounter                  ** (%C71) Piercing counter
norescounter:

*********************************************************************
* Wrong selection option protection

* no piercing option,no lead in option or worklist enabled reset all pre piercing
* if origin 19 selected, disable all option

CAL  RTRIG_NOPIERC (CLK:=EnNoPiercing) ** (%rLsGui29.5) No piercing execution
CAL  RTRIG_NOLEAD (CLK:=EnNoLeadIn) ** (%rLsGui29.6) No lead-in execution
CAL  RTRIG_WORK_ENAB (CLK:=WorkListEnabled) ** (LSRPlcOp0.5) Worklist mode enabled
CAL  RTRIG_ORIG19 (CLK:=VisLedOrigGui.19)         * Origin 19 selected
CAL  RTRIG_BLOCK_S (CLK:=BUP_BLKSRC) ** ui16.24 Selezione esecuzione ricerca blocco

LD   RTRIG_NOPIERC.Q
OR   RTRIG_NOLEAD.Q
OR   RTRIG_WORK_ENAB.Q
OR   VisLedOrigGui.19                             * Origin 19 selected
OR   RTRIG_BLOCK_S.Q
JMPCN resAllpierc

LD   ALWAYS_ONE                    ** PLCFLAGS.1  Flag sempre stato on
R    AllPrePiercing                ** (%rLsGui29.7) Force all pre-piercing

resAllpierc:

* All piercing option reset no pierc and no lead in

CAL  RTRIG_ALLPIERC (CLK:=AllPrePiercing) ** (%rLsGui29.7) Force all pre-piercing

LD   RTRIG_ALLPIERC.Q
OR   VisLedOrigGui.19                             * Origin 19 selected
OR   RTRIG_BLOCK_S.Q
JMPCN resNopierc

LD   ALWAYS_ONE                    ** PLCFLAGS.1  Flag sempre stato on
R    EnNoPiercing                  ** (%rLsGui29.5) No piercing execution
R    EnNoLeadIn                    ** (%rLsGui29.6) No lead-in execution

resNopierc:

* Stop end track geometry reset stop end piece

CAL  RTRIG_RES_PIECE (CLK:=StopEndTrackGeometry) ** (LSRPlcOp0.7) stop at the end of the track/geometry

LD   RTRIG_RES_PIECE.Q
OR   VisLedOrigGui.19                             * Origin 19 selected
OR   RTRIG_BLOCK_S.Q
JMPCN no_res_endpiece

LD   ALWAYS_ONE                    ** PLCFLAGS.1  Flag sempre stato on
R    StopEndPiece                  ** (LSRPlcOp0.19) stop at the end of the piece

no_res_endpiece:

* Stop end piece reset stop end Stop End Track Geometry

CAL  RTRIG_RES_GEOM  (CLK:=StopEndPiece) ** (LSRPlcOp0.19) stop at the end of the piece

LD   RTRIG_RES_GEOM.Q
****OR   VisLedOrigGui.19                             * Origin 19 selected
OR   RTRIG_BLOCK_S.Q
JMPCN  no_res_end_geometr

LD   ALWAYS_ONE                    ** PLCFLAGS.1  Flag sempre stato on
R    StopEndTrackGeometry          ** (LSRPlcOp0.7) stop at the end of the track/geometry

no_res_end_geometr:

CAL  FTRIG_RES_AUTO_CLEAN (CLK:=NozzleCleanPresent) ** (LSRPlcOp1.5) Nozzle clean active

LD   FTRIG_RES_AUTO_CLEAN.Q
OR   VisLedOrigGui.19                             * Origin 19 selected
OR   RTRIG_BLOCK_S.Q
JMPCN res_auto_clean

LD   ALWAYS_ONE                    ** PLCFLAGS.1  Flag sempre stato on
R    AutoNozzleClean               ** (%rLsGui29.9) Nozzle clean active

res_auto_clean:

********************************************************************************
* DB Laser upload synchronism (no_usr db present)
********************************************************************************

*LD   %Uipl.CurPsw                * Valore corrente Password Attiva
*EQ   255
*ST   UseDbUser                   *(LsPlc0.5) User db is used online db

**********************************************************************
* Clear alarm function
**********************************************************************
LD  ButtClearAlarm                 ** (gGui23.0) Clear alarm interface push-button
OR  RemContrCancAlarm			   * Xhc_Puls.31 Clear alarm
AND (
LD  PRGSTOP_CN0                    ** (cn0.rc8.1)  Programma interrotto CN0
ORN PRGRUN_CN0                     ** M0.0 cn0.rc8.0  Programma in corso
)
JMPCN noClearAlarm

LD   0
ST   %PLCerr0
ST   %PLCerr1
ST   %PLCerr2
ST   %PLCerr3
ST   %PLCerr4
ST   %PLCerr5
ST   %PLCerr6
ST   %PLCerr7
ST   %PLCerr8
ST   %PLCerr20
ST   %PLCerr21

ST   %PLCmsg0
ST   %PLCmsg1
ST   %PLCmsg2
ST   %PLCmsg3
ST   %PLCmsg4
ST   %PLCmsg5
ST   %PLCmsg6
ST   %PLCmsg7

noClearAlarm:

**@@@ OUT_TEST    * Digital Outputs test management

END_FUNCTION

(* ---- Log.plc ---- *)
*******************************************************************************
*   Log
*   ESAutomotion
*   LASER machine
*   Time Logger
*******************************************************************************

#include "Iol.inc"
#include "LsrGest.inc"

VAR

R_TRIG_COUNT:               R_TRIG;
R_TRIG_COUNT1:              R_TRIG;
R_TRIG_COUNT2:              R_TRIG;
R_TRIG_COUNT4:              R_TRIG;

RTRIG_1:                    R_TRIG;
RTRIG_2:                    R_TRIG;
RTRIG_3:                    R_TRIG;
FTRIG_4:                    F_TRIG;
RTRIG_5:                    R_TRIG;
RTRIG_6:                    R_TRIG;
RTRIG_7:                    R_TRIG;
RTRIG_8:                    R_TRIG;
RTRIG_9:                    R_TRIG;
RTRIG_10:                   R_TRIG;
RTRIG_11:                   R_TRIG;
RTRIG_12:                   R_TRIG;
RTRIG_13:                   R_TRIG;
RTRIG_14:                   R_TRIG;
RTRIG_15:                   R_TRIG;
RTRIG_16:                   R_TRIG;
RTRIG_17:                   R_TRIG;
RTRIG_18:                   R_TRIG;
RTRIG_19:                   R_TRIG;
RTRIG_20:                   R_TRIG;
FTRIG_21:                   F_TRIG;
RTRIG_22:                   R_TRIG;
FTRIG_23:                   F_TRIG;
FTRIG_24:                   F_TRIG;
RTRIG_25:                   R_TRIG;
FTRIG_26:                   F_TRIG;
RTRIG_27:                   R_TRIG;
FTRIG_28:                   F_TRIG;

FTRIG_DEL_LOGCNC:           F_TRIG;

jogp:                       BOOL;            * Positive command movement
jogm:                       BOOL;            * Negative command movement
jog_mov:                    BOOL;            * Jog in progress
END_VAR

VAR_IN_OUT
#include "mem.inc"
END_VAR

FUNCTION  LOG

* Function for diary ***

* Total Machine Time

CAL R_TRIG_COUNT2 (CLK:=%PLCFLAGS.10)

LD   R_TRIG_COUNT2.Q
JMPCN no_inc1

LD  Count_sec_tot                  ** (rLsPlc46) Counter for second, total time
ADD 1
ST  Count_sec_tot                  ** (rLsPlc46) Counter for second, total time

no_inc1:

LD   Count_sec_tot                 ** (rLsPlc46) Counter for second, total time
EQ   86400
JMPCN no_update_day_tot
LD   0
ST   Count_sec_tot                 ** (rLsPlc46) Counter for second, total time

LD   Count_day_tot                 ** (rLsPlc44) Counter for day, total time
ADD  1
ST   Count_day_tot                 ** (rLsPlc44) Counter for day, total time
no_update_day_tot:

LD   Count_day_tot                 ** (rLsPlc44) Counter for day, total time
EQ   365
JMPCN no_update_year

LD   0
ST   Count_day_tot                 ** (rLsPlc44) Counter for day, total time

LD   Count_year_tot                ** (rLsPlc45) Counter for years, total time
ADD  1
ST   Count_year_tot                ** (rLsPlc45) Counter for years, total time

no_update_year:
*

* Time from last switch-on

CAL R_TRIG_COUNT (CLK:=%PLCFLAGS.8)

LD  R_TRIG_COUNT.Q
JMPCN no_reset_timer

LD  0
ST  Count_sec_day                  ** (rLsPlc40) Counter for second, last switch on
ST  Count_day_day                  ** (rLsPlc41) Counter for day, last switch on

no_reset_timer:

CAL R_TRIG_COUNT1 (CLK:=%PLCFLAGS.10)

LD   R_TRIG_COUNT1.Q
JMPCN no_inc

LD  Count_sec_day                  ** (rLsPlc40) Counter for second, last switch on
ADD 1
ST  Count_sec_day                  ** (rLsPlc40) Counter for second, last switch on

no_inc:

LD   Count_sec_day                 ** (rLsPlc40) Counter for second, last switch on
EQ   86400
JMPCN no_update_day
LD   0
ST   Count_sec_day                 ** (rLsPlc40) Counter for second, last switch on

LD   Count_day_day                 ** (rLsPlc41) Counter for day, last switch on
ADD  1
ST   Count_day_day                 ** (rLsPlc41) Counter for day, last switch on
no_update_day:
*

* Total time laser On

CAL  R_TRIG_COUNT4 (CLK:=%PLCFLAGS.10)

LD   R_TRIG_COUNT4.Q
AND  (
LD   HW_PWM_CFG_FC                           ** Laser I/F board PWM_CFG register: FC
OR   INP_flyCutModeON                        ** application turn flyCut mode ON
)
JMPCN no_inc2

LD   Count_sec_lson                ** (rLsPlc47) Counter for second, Laser on
ADD  1
ST   Count_sec_lson                ** (rLsPlc47) Counter for second, Laser on

no_inc2:

LD   Count_sec_lson                ** (rLsPlc47) Counter for second, Laser on
EQ   86400
JMPCN no_day_inc

LD   0
ST   Count_sec_lson                ** (rLsPlc47) Counter for second, Laser on

LD   Count_day_lason               ** (rLsPlc48) Counter for day, laser on
ADD  1
ST   Count_day_lason               ** (rLsPlc48) Counter for day, laser on
no_day_inc:

*
******************************************************************************************
* Log Log.cfs

LD   %ax27.ra0.8                             * Positive command movement
OR   %ax28.ra0.8                             * Positive command movement
OR   %ax29.ra0.8                             * Positive command movement
OR   %ax30.ra0.8                             * Positive command movement
OR   %ax51.ra0.8                             * Positive command movement
OR   %ax52.ra0.8                             * Positive command movement
OR   %ax53.ra0.8                             * Positive command movement
AND  ch0_InJOG                     ** %cn0.rc0.9 CH0 en Modo JOG
ST   jogp                          ** Positive command movement

CAL  RTRIG_1(CLK:=jogp)            ** Positive command movement
LD   RTRIG_1.Q
S    LogVarPlc.0                             * Jog + Command

LD   %ax27.ra0.9                             * Negative command movement
OR   %ax28.ra0.9                             * Negative command movement
OR   %ax29.ra0.9                             * Negative command movement
OR   %ax30.ra0.9                             * Negative command movement
OR   %ax51.ra0.9                             * Negative command movement
OR   %ax52.ra0.9                             * Negative command movement
OR   %ax53.ra0.9                             * Negative command movement
AND  ch0_InJOG                     ** %cn0.rc0.9 CH0 en Modo JOG
ST   jogm                          ** Negative command movement

CAL  RTRIG_2(CLK:=jogm)            ** Negative command movement

LD   RTRIG_2.Q
S    LogVarPlc.1                             * Jog - Command

CAL  RTRIG_3(CLK:=Pul_Start)       ** (gPlc0.1)Start pushbutton

LD   RTRIG_3.Q
S    LogVarPlc.2                             * Program Start

CAL  FTRIG_4(CLK:=ch0_InRun)       ** %cn0.rc8.0 CH0 Programa RUN activo

LD   FTRIG_4.Q
S    LogVarPlc.3                             * Program Fineshed

CAL  RTRIG_5(CLK:=ch0_InRun)       ** %cn0.rc8.0 CH0 Programa RUN activo

LD   RTRIG_5.Q
S    LogVarPlc.4                             * Program in Run

CAL  RTRIG_6(CLK:=Pul_Stop)        ** (gPlc0.2)Stop pushbutton

LD   RTRIG_6.Q
S    LogVarPlc.5                             * Stop button pushed

CAL  RTRIG_7(CLK:=ch0_InHold)      ** %cn0.rc8.1 CH0 Programa RUN con HOLD activo

LD   RTRIG_7.Q
S    LogVarPlc.6                             * Program in hold

CAL  RTRIG_8(CLK:=Pul_Reset)       ** (gPlc0.3)Reset pushbutton

LD   RTRIG_8.Q
S    LogVarPlc.7                             * Reset button pushed

CAL  RTRIG_9(CLK:=SparoMan_On)     ** (LsGui0.10) Sparo Manuale Start

LD   RTRIG_9.Q
S    LogVarPlc.8                             * Manual Laser Shot Start Button

CAL  RTRIG_10(CLK:=SparoMan_Stop)  ** (LsGui0.11) Sparo Manuale Stop

LD   RTRIG_10.Q
S    LogVarPlc.9                             * Manual Laser Shot Stop Button

CAL  RTRIG_11(CLK:=GAS_test)       	 ** M107.0 Test gas in progress for prop. valve

LD   RTRIG_11.Q
S    LogVarPlc.10                            * Start gas test

CAL  RTRIG_12(CLK:=O_O_EV_OPEN_N2)		 ** Elettrovalvola apertura Azoto

LD   RTRIG_12.Q
S    LogVarPlc.11                            * N2 Open

CAL  RTRIG_13(CLK:=O_O_EV_OPEN_O2) ** Elettrovalvola apertura Ossigeno

LD   RTRIG_13.Q
S    LogVarPlc.12                            * O2 Open

CAL  RTRIG_14(CLK:=O_O_EV_OPEN_ARIA)		 ** Elettrovalvola apertura Aria taglio

LD   RTRIG_14.Q
S    LogVarPlc.13                            * Air Open

CAL  RTRIG_15(CLK:=PLC_SEL_REF)    ** ui16.1 Selezione Modo REF da Plc

LD   RTRIG_15.Q
S    LogVarPlc.14                            * Reference mode

CAL  RTRIG_16 (CLK:=PLC_SEL_JOG)   ** ui16.2 Selezione Modo JOG da Plc

LD   RTRIG_16.Q
S    LogVarPlc.15                            * Jog Mode

CAL  RTRIG_17 (CLK:=PLC_SEL_INC)   ** ui16.3 Selezione Modo INC da Plc

LD   RTRIG_17.Q
S    LogVarPlc.16                            * Incremental Mode

CAL  RTRIG_18 (CLK:=PLC_SEL_MDI)   ** ui16.4 Selezione Modo MDI da Plc

LD   RTRIG_18.Q
S    LogVarPlc.17                            * MDI Mode

CAL  RTRIG_19 (CLK:=PLC_SEL_AUT)   ** ui16.5 Selezione Modo AUT da Plc

LD   RTRIG_19.Q
S    LogVarPlc.18                            * Auto Mode

CAL  RTRIG_20 (CLK:=%PlcOp0.2)     ** DryRun

LD   RTRIG_20.Q
S    LogVarPlc.19                            * Dry Run Enable

CAL  FTRIG_21 (CLK:=%PlcOp0.2)     ** DryRun

LD   FTRIG_21.Q
S    LogVarPlc.20                            * Dry Run Disable

CAL  RTRIG_22 (CLK:=%LSRPlcOp0.6)            ** Macchina in modo Dry Run

LD   RTRIG_22.Q
S    LogVarPlc.21                            * Force Z Up Enable

CAL  FTRIG_23 (CLK:=%LSRPlcOp0.6)            ** Macchina in modo Dry Run

LD   FTRIG_23.Q
S    LogVarPlc.22                            * Force Z up Disable

LD   jogp                          ** Positive command movement
OR   jogm                          ** Negative command movement
ST   jog_mov                       ** Jog in progress

CAL  FTRIG_24 (CLK:=jog_mov)       ** Jog in progress

LD   FTRIG_24.Q
S    LogVarPlc.23                            * Jog Movement Stop

CAL  RTRIG_25 (CLK:=%LSRPlcOp0.8)  ** Z axis in simulation (always in UP position)

LD   RTRIG_25.Q
S    LogVarPlc.24                            * No Z axis movement Enable

CAL  FTRIG_26 (CLK:=%LSRPlcOp0.8)  ** Z axis in simulation (always in UP position)

LD   FTRIG_26.Q
S    LogVarPlc.25                            * No Z axis movement disable

CAL  RTRIG_27 (CLK:=EnableSheetCont) ** (gGui0.6) Enable sheet control dimension

LD   RTRIG_27.Q
S    LogVarPlc.26                            * Enable sheet control dimension

CAL  FTRIG_28 (CLK:=EnableSheetCont) ** (gGui0.6) Enable sheet control dimension

LD   FTRIG_28.Q
S    LogVarPlc.27                            * Disable sheet control dimension

CAL  FTRIG_DEL_LOGCNC (CLK:=IntCopyLogg) ** ui39.0 interface signal for log transfer from cnc to pc folder

LD   FTRIG_DEL_LOGCNC.Q
S    LogVarPlc.31                            * Delete log file content

*******************************************************************************************
END_FUNCTION

(* ---- lubr.plc ---- *)
*******************************************************************************
*   LUBR.PLC
*   ESAutomotion
*   LASER machine
*******************************************************************************
VAR
#include "Cnc.inc"
END_VAR

VAR_IN_OUT
#include "mem.inc"
END_VAR

#include "Iol.inc"

VAR
TON_PUMP_ON_MINUTE:    TON;
TON_PUMP_ON_HOUR:      TON;
TON_REST_PUMP:         TON;
TON_REST_PUMP1:        TON;
TON_REST_PUMP2:        TON;
TON_REST_PUMP3:        TON;
appoggio:             BOOL;
TurnPumpTMP:          BOOL;
RestartPump:          BOOL;

RTRIG_TIME:         R_TRIG;
RTRIG_PUMP:         R_TRIG;
RTRIG_PUMP2:         R_TRIG;

Hour_axes_mov       AT %LsGui5;       * (LsGui5) Hour axes movement
Minute_axes_mov     AT %LsGui6;       * (LsGui6) Minute axes movement

hour                AT %rLsPlc23;     * (rLsPlc23) timer for lubrication cycle minute
timer_minute        AT %rLsPlc24;     * (rLsPlc24) time minutes
timer_hour          AT %rLsPlc25;     * (rLsPlc25) time hour
pump_on_time        AT %rLsPlc26;     * (rLsPlc26) pump on period [s]
pump_off_time        AT %rLsPlc35;     * (rLsPlc35) pump off time [s]
Repetition           AT %rLsPlc37;     * (rLsPlc37)

PumpCount:            DWORD;
END_VAR

VAR_IN_OUT
PulLubr             AT %LsGui4.0;     * (LsGui4.0) Push Button manual lubrication
TurnPump            AT %LsGui4.1;     * (LsGui4.1) Turn on pump
MinLevel            AT %LsGui4.2;     * (LsGui4.2) Min level in lubrication system
MinPressure         AT %LsGui4.3;     * (LsGui4.3) Min pressure in lubrication system
END_VAR

******************************************************************************
*   Lubrication management
******************************************************************************
FUNCTION Lubrication

LDN  %ax27.ra3.0                      * axis not move
ORN  %ax30.ra3.0                      * axis not move
ORN  %ax28.ra3.0                      * axis not move
ORN  %ax31.ra3.0                      * axis not move
ORN  %ax36.ra3.0                      * axis not move
ST   appoggio

CAL  RTRIG_TIME(CLK:=%PLCFLAGS.10)

***************************************
LD   RTRIG_TIME.Q
AND  appoggio
JMPCN no_count
LD   second                        ** (rLsPlc21) timer for lubrication cycle second
ADD  1
ST   second                        ** (rLsPlc21) timer for lubrication cycle second
no_count:

LD   second                        ** (rLsPlc21) timer for lubrication cycle second
EQ   60
JMPCN inc_minut
LD   minute                        ** (rLsPlc22) timer for lubrication cycle minute
ADD  1
ST   minute                        ** (rLsPlc22) timer for lubrication cycle minute

LD   0
ST   second                        ** (rLsPlc21) timer for lubrication cycle second
inc_minut:

LD   minute                        ** (rLsPlc22) timer for lubrication cycle minute
EQ   60
JMPCN inc_hour
LD   hour                          ** (rLsPlc23) timer for lubrication cycle minute
ADD  1
ST   hour                          ** (rLsPlc23) timer for lubrication cycle minute

LD   0
ST   minute                        ** (rLsPlc22) timer for lubrication cycle minute
inc_hour:

***************************************
LD  %LSRPlcOp1.13                  ** Enable lubrication by minute, default by hour
JMPCN no_lubr_by_minute

LD   minute                           * (rLsPlc22) timer for lubrication cycle second
GE   timer_minute                      * (rLsPlc24) time minutes
ANDN RestartPump
ST   TurnPumpTMP                      * pump on by automatic cycle

LD   PulLubr                          * (LsGui4.0) Push Button manual lubrication
ST   TurnPump                         * (LsGui3.0) Turn on pump

CAL  TON_PUMP_ON_MINUTE (IN:=TurnPumpTMP,PT:=pump_on_time)
CAL  TON_REST_PUMP (IN:=TON_PUMP_ON_MINUTE.Q,PT:=pump_off_time)

LD   TON_REST_PUMP.Q
ST   RestartPump

LD   TON_PUMP_ON_MINUTE.Q
JMPCN res_timer_pump1

LD   ALWAYS_ZERO
ST   TurnPumpTMP                      * pump on by automatic cycle

LD   PumpCount
GE   Repetition
JMPCN no_res_pump

 LD   0
 ST   PumpCount

 LD   0
 ST   minute                           * (rLsPlc22) timer for lubrication cycle second
no_res_pump:

res_timer_pump1:

CAL  RTRIG_PUMP (CLK:=TurnPumpTMP)

LD   RTRIG_PUMP.Q
JMPCN no_inc_pump

LD   PumpCount
ADD  1
ST   PumpCount

no_inc_pump:

LD   PulLubr                          * (LsGui4.0) Push Button manual lubrication
OR   TurnPumpTMP                      * pump on by automatic cycle
ST   TurnPump                         * (LsGui3.0) Turn on pump

no_lubr_by_minute:
LDN  %LSRPlcOp1.13                 ** Enable lubrication by minute, default by hour
JMPCN no_lubr_by_hour

LD   hour                             *(rLsPlc23) timer for lubrication cycle hour
GE   timer_hour                       * (rLsPlc25) time hour
ANDN RestartPump
ST   TurnPumpTMP                      * pump on by automatic cycle

CAL  TON_PUMP_ON_HOUR (IN:=TurnPumpTMP,PT:=pump_on_time)
CAL  TON_REST_PUMP2 (IN:=TON_PUMP_ON_HOUR.Q,PT:=pump_off_time)

LD   TON_REST_PUMP2.Q
ST   RestartPump

LD   TON_PUMP_ON_HOUR.Q
JMPCN res_timer_pump2

LD   ALWAYS_ZERO
ST   TurnPumpTMP                      * pump on by automatic cycle

LD   PumpCount
GE   Repetition
JMPCN no_res_pump2

 LD   0
 ST   PumpCount

 LD   0
 ST   hour                             *(rLsPlc23) timer for lubrication cycle hour
no_res_pump2:

res_timer_pump2:

CAL  RTRIG_PUMP2 (CLK:=TurnPumpTMP)

LD   RTRIG_PUMP2.Q
JMPCN no_inc_pump2

LD   PumpCount
ADD  1
ST   PumpCount

no_inc_pump2:

LD   PulLubr                          * (LsGui4.0) Push Button manual lubrication
OR   TurnPumpTMP                      * pump on by automatic cycle
ST   TurnPump                         * (LsGui3.0) Turn on pump

no_lubr_by_hour:

***************************************
LD   I_I_LUB_LOW_LEVEL             ** Lubrication: low oil level
ST   MinLevel                      ** (LsGui4.2) Min level in lubrication system
ST   %PLCmsg4.27                      * Lubrication system low level

LD   I_I_LUB_LOW_PRESSURE             ** Lubrication: low oil pressure
ST   MinPressure                     ** (LsGui4.3) Min pressure in lubrication system
ST   %PLCmsg4.28                      * Lubrication system low pressure

LD   TurnPump                      ** (LsGui4.1) Turn on pump
ST   O_O_LUB                       ** Lubrication

LD   hour                          ** (rLsPlc23) timer for lubrication cycle minute
ST   Hour_axes_mov                 ** (LsGui5) Hour axes movement

LD   minute                        ** (rLsPlc22) timer for lubrication cycle minute
ST   Minute_axes_mov               ** (LsGui6) Minute axes movement

END_FUNCTION

(* ---- LuciMacc.plc ---- *)
*******************************************************************************
*   LUCIMACC.PLC
*   ESAutomotion
*   LASER machine
*******************************************************************************
VAR
#include "Cnc.inc"

Macchina_in_ANOMALIA:       BOOL;   ** Macchina in anomalia
Macchina_in_HOLD_oper:      BOOL;   ** Macchina in hold operatore
Macchina_in_lavorazione:    BOOL;   ** Macchina in lavorazione
END_VAR

VAR_IN_OUT
#include "mem.inc"
END_VAR

#include "Iol.inc"

*******************************************************************************
*    * Gestione Lampade Macchina
*******************************************************************************
FUNCTION LuciMacc

*******************************************************************************
*   Illuminazione CABINA
*******************************************************************************
LD   ON_OFF_CABINA                 ** (LsGui0.1)
ST	 O_O_LUCE_CABINA                ** machine light

*******************************************************************************
*   Illuminazione Testa Laser
*******************************************************************************
LD   ON_OFF_TESTA_LASER            ** (LsGui0.2)
ST   O_O_LUCE_SU_TESTA_LASER       ** head light

*******************************************************************************
* Macchina in ANOMALIA
*******************************************************************************
LDN  O_O_CNC_OK                    ** CNC OK
OR   ALARM_ACT		                   ** M100.3  Allarme attivo
ST	 Macchina_in_ANOMALIA

*******************************************************************************
* Macchina in HOLD operatore
*******************************************************************************
LD   PRGSTOP_CN0		                 ** (cn0.rc8.1)  Programma interrotto CN0
ANDN Macchina_in_ANOMALIA	** Macchina in anomalia
ST	 Macchina_in_HOLD_oper	** Macchina in hold operatore

*******************************************************************************
* Macchina in ciclo senza allarmi e no hold
*******************************************************************************
LD   MACCH_IN_AUTO		               ** M100.25 SELEZIONE MACCHINA IN AUTOMATICO
AND	 PRGRUN_CN0 		                 ** M0.0 cn0.rc8.0  Programma in corso
ANDN Macchina_in_HOLD_oper
ANDN Macchina_in_ANOMALIA
ST	 Macchina_in_lavorazione

*******************************************************************************
*   Colonnina luminosa: Luce ROSSA
*******************************************************************************
LDN  EMERGENZA_PLC_CN     		       ** M100.0  Emergenza da PLC o da CN
*OR   NORMAL_BLINK     		           ** PLCFLAGS.10 Lampeggio normale (0.5 sec.)
ANDN MACCHINA_OK			                ** M100.1  Macchina OK
OR(
LD   MACCHINA_OK			                ** M100.1  Macchina OK
AND	 Macchina_in_ANOMALIA		** Macchina in anomalia
*AND  NORMAL_BLINK     		           ** PLCFLAGS.10 Lampeggio normale (0.5 sec.)
)
ST   O_O_LAMPADA_ROSSA	            ** Red lamp

*******************************************************************************
* Colonnina luminosa: Luce VERDE
*******************************************************************************
LD   Macchina_in_lavorazione		** Macchina in lavorazione
*AND  NORMAL_BLINK     		           ** PLCFLAGS.10 Lampeggio normale (0.5 sec.)
ORN	 Macchina_in_lavorazione		** Macchina in lavorazione
AND	 MACCHINA_OK			                ** M100.1  Macchina OK
ANDN Macchina_in_ANOMALIA		** Macchina in anomalia
AND  PRGRUN_CN0 			                ** M0.0 cn0.rc8.0  Programma in corso
ST	 O_O_LAMPADA_VERDE	             ** Green lamp

*******************************************************************************
* Colonnina luminosa: Luce ARANCIO
*******************************************************************************
*LD   MACCH_IN_AUTO			              ** M100.25 SELEZIONE MACCHINA IN AUTOMATICO YANG
LDN PRGRUN_CN0 			                ** M0.0 cn0.rc8.0  Programma in corso
OR	 Macchina_in_HOLD_oper		** Macchina in hold operatore
*AND	 NORMAL_BLINK			               ** PLCFLAGS.10 Lampeggio normale (0.5 sec.)
ANDN Macchina_in_ANOMALIA		** Macchina in anomalia
AND	 MACCHINA_OK			                ** M100.1  Macchina OK
ST	 O_O_LAMPADA_ARANCIONE	         ** Orange lamp

END_FUNCTION

(* ---- MainFast.plc ---- *)
*******************************************************************************
*   MAIN FAST UNIFIED
*   ESAutomotion
*   LASER machine
*******************************************************************************
#funcdec "intgraph.plc"
#funcdec "DynMng.plc"

VAR

#include "MainFast.inc"
#include "Iof.inc"
Appoggio:           BOOL;
TP_PGMSEND:         TP;
F_TRIG_PGMSEND:     F_TRIG;
TP_PGMSEND_1:       TP;
F_TRIG_PGMSEND_1:   F_TRIG;
R_TRIG_FOLLOW:      R_TRIG;

analize_solder:     BOOL;       * x gestione analizza eventi sensore
cax_ini_solder:     DWORD;      * quota asse C campionata inizio di una saldatura
ofs_center_solder:  DWORD;      * offset del centro della saldatura
ResultFir3:         DWORD;
cn0_rc129:          DWORD;
cn0_rc129_filtered: DWORD;

cap_temp:           DWORD;       * Test RTCP con capacitivo
cap_fir_time:       DWORD;       * Test RTCP con capacitivo
vectorSelect:       DWORD;       * vectorSelect 1 = tool, 2 = surface, 6 = Z
END_VAR

VAR_IN_OUT
#include "mem.inc"
TovisualizeWiget    AT %HMI_ONE.mcp_in.28;
EnBvlConerOptim     AT %HMI_ONE.mcp_in.29;
CornerChangeCmd     AT %HMI_ONE.mcp_in.30;
END_VAR

#include "Iol.inc"
#include "LsrGest.inc"

*******************************************************************************
*   MainFast
*******************************************************************************
FUNCTION MAIN

LD   %LSRCostK31                   ** Capacitive sensor range
DIV  10
ST   MaxVolt_x100
LD   4095
ST   MaxADCPoints

**************************************************
*   FIR on capacitive for RTCP test
**************************************************
LD   %cn0.rc0.12                    * CN0 in auto mode
OR   PRGRUN_CN0                    ** M0.0 cn0.rc8.0  Programma in corso
OR   %PLCFLAGS.8                    * one scan
ST   appoggio

CAL  RT_PRGRUN(CLK=appoggio)

LD   RT_PRGRUN.Q
JMPCN no_init_fir

LD   100                            * 100 msec filtro fisso per gestione test RTCP
DIV  %plc0.PlcCycle
ST   cap_fir_time

LD   0
FIR_INIT (INS=8, LEN=cap_fir_time)
ST   error1     * 0 = OK

no_init_fir:
**************************************************
*   FIR on %cn0.rc129 (CO_TOOL_SURFACE_ANGLE)
**************************************************
LD   %uvHeads0.uvhCommand[0].1          * UVH_COMMAND_PLC_VRTC_HANDLING
JMPC vrtc_handling

LD   %TsCutDataLinear.CDL_rpar0
DIV  %plc0.PlcCycle
ST   fir_time

LD   0
FIR_INIT (INS=3, LEN=fir_time)
ST   error1     * 0 = OK

vrtc_handling:
**************************************************
*   Define angle management about
*   setpoint and feedback of VRTC
**************************************************
LD   0
ST   bevAngleHead1_calc1
ST   bevAngleHead1_calc2
ST   bevAngleHead1_calc3

LD   %uvHeads0.uvhCommand[0].1          * UVH_COMMAND_PLC_VRTC_HANDLING
JMPCN no_vrtc_handling

LD   %cn0.rc129                         * CO_TOOL_SURFACE_ANGLE
ST   cn0_rc129
ST   cn0_rc129_filtered

LD   0                       * N/C
FIR_RUN (INS=3, X=cn0_rc129)
ST   ResultFir3

LD   ResultFir3                       ** Result
EQ   2147483647
JMPC fir3_err

LD   ResultFir3
ST   cn0_rc129_filtered

fir3_err:
LD   %uvHeads0.uvhSurfaceCommand3
ST   vectorSelect

LD   vectorSelect                  * Pipe cutting: 1 = tool, 2 = surface, 6 = Z
EQ   1
JMPCN reg_0

LD   0
ST   bevAngleHead1_calc1
ST   bevAngleHead1_calc2
JMP  reg_com

reg_0:
LD   vectorSelect                  * Pipe cutting: 1 = tool, 2 = surface, 6 = Z
EQ   6
JMPCN reg_1

LD   %cn0.rc128                         * CO_TOOL_Z_ANGLE
ST   bevAngleHead1_calc1
ST   bevAngleHead1_calc2
JMP  reg_com

reg_1:
LD   cn0_rc129_filtered
***LD   0                               * Da usare per G2-G3 !!!
ST   bevAngleHead1_calc1
ST   bevAngleHead1_calc2

reg_com:

****************************************
*   Patch per OMP !
*   Richiesta di OMP per regolazione
*   lungo l'utensile !
****************************************
LD   vectorSelect                  * Pipe cutting: 1 = tool, 2 = surface, 6 = Z
EQ   1
JMPCN reg_end_omp

LD   cn0_rc129_filtered
***LD   0                               * Da usare per G2-G3 !!!
ST   bevAngleHead1_calc1
ST   bevAngleHead1_calc3

LD   0
ST   bevAngleHead1_calc2

reg_end_omp:

no_vrtc_handling:

**************************************************
* Tcp position
**************************************************
LD   PRGRUN_CN0
OR   PLC_SEL_JOG
OR   PLC_SEL_AUT
ST   appoggio

CAL  RTRIG_INIT (CLK:=appoggio)

LD   RTRIG_INIT.Q
JMPCN no_init

LD      0               * N/C
WJS_LOAD (INS=6,CH=3,TWI=1,THD=1,CED=1,SVL=0,CHX=0,CHY=1,CHZ=2,CHA=0,CHB=0,FRX=0,FRY=0,FRZ=0,FOX=0,FOY=0,FOZ=0)
WJS_LOAD (INS=7,CH=0,TWI=1,THD=1,CED=1,SVL=0,CHX=16#40000000,CHY=16#40000001,CHZ=16#40000002,CHA=0,CHB=0,FRX=0,FRY=0,FRZ=0,FOX=0,FOY=0,FOZ=0) * TODO!
***WJS_LOAD (INS=7,CH=3,TWI=1,THD=1,CED=1,SVL=0,CHX=16#40000000,CHY=16#40000001,CHZ=16#40000002,CHA=16#40000000,CHB=16#40000000,FRX=0,FRY=0,FRZ=0,FOX=0,FOY=0,FOZ=0) * TODO!
ST   loadconfig             * 0 = OK

no_init:
LD      loadconfig
NE      0
JMPC    errorAngle

LD      0               * N/C
WJS_BEAM_CALC (INS=6,SVL=0)
WJS_BEAM_CALC (INS=7,SVL=0)
ST      calcBeam            * 0 = OK

LD      calcBeam
NE      0
JMPC    errorAngle

LD   0
WJS_GETX_TCP (INS=6)
ST   tcp_X_head1_fast
LD   0
WJS_GETY_TCP (INS=6)
ST   tcp_Y_head1_fast
LD   0
WJS_GETZ_TCP (INS=6)
ST   tcp_z

LD      tcp_z
EQ      2147483647
JMPC    errorAngle

LD      tcp_z
ST      tcp_Z_head1_fast                      * (C152) z tcp of head 1

JMP  errorTCPz
errorAngle:
LD      0
ST      tcp_Z_head1_fast                      * (C152) z tcp of head 1
errorTCPz:

* TODO!
***LD   %ax34.ra4
***ST   %C159

* TODO!
***LD   0
***WJS_GETX_TCP (INS=7)
***ST   %C160
***LD   0
***WJS_GETY_TCP (INS=7)
***ST   %C161
***LD   0
WJS_GETZ_TCP (INS=7)
ST   %C162

* TODO!
***LD   %ax34.ra24
***ST   %C163

**************************************************
*   @@@ START = SIMULATION
**************************************************
LD   %M33                  ** PLC SIMULATION !
EQ   1
JMPCN NoSIM

FAST_SIM
JMP EndFast

NoSIM:
FAST_REAL

EndFast:

LD   0                       * N/C
FIR_RUN (INS=8, X=%C120)     * Capacitivo (ADC) NON linearizzato
ST   cap_temp

LD   cap_temp
EQ   2147483647
JMPC err_fir

LD   cap_temp
ST   IA_A18_19_DIST_LINEAR_FIR

err_fir:

**************************************************
LD   Gest5Ax
AND(
     LD   gG800GStatus
     GT   0
)
JMPCN _AssignAng5x
     LD   Capacit_Anal
     MUL  1000
     DIV (
     LD   bevAngleHead1_calc3
     COS
     )
     ST   %C121               * (C121) Logical resource VRTC1 (surface)

     LD   Capacit_Anal
     MUL  1000
     DIV (
     LD   bevAngleHead1_calc1
     COS
     )
     ST  %C131                * (C131) Logical resource VRTC0 (tool)

	 ***************************************
     *   Normalizzazione capacitivo
     *   come altezza di taglio in mm
     ***************************************
     LD   Capacit_Anal                  ** (C102)Analogica Capacitivo
     MUL  MaxVolt_x100
     MULDIV (M=10000, D=MaxADCPoints)
     DIV  (
     LD   bevAngleHead1_calc1
     COS
     )
     DIV  10                             * Per visualizzare due cifre decimali
     ST   Capacit_Anal_Mm		             ** (C103)Analogica Capacitivo in mm

JMP _AssignAngCom
_AssignAng5x:
     LD   Capacit_Anal
     ST   %C121               * (C121) Logical resource VRTC1 (surface)

     LD   Capacit_Anal
     ST   %C131               * (C131) Logical resource VRTC0 (tool)

	 LD   Capacit_Anal                  ** (C102)Analogica Capacitivo
     MUL  MaxVolt_x100
     MULDIV (M=10000, D=MaxADCPoints)
     DIV  1000
     DIV  10                             * Per visualizzare due cifre decimali
     ST   Capacit_Anal_Mm		             ** (C103)Analogica Capacitivo in mm

_AssignAngCom:

***************************************
*   Sicurezza
***************************************
LD   CUT_DISTANCE
DIV  10
ADD  25                            *  RANGE
ST   StandOff                      ** Valore distanza taglio in centesimi

LD   BlcAvX1_Sens_Capac            ** M74.3 Blocco avanz. asse X1 Sens. Capacitivo in contatto con la lamiera
OR   BlcAvY1_Sens_Capac            ** M74.6 Blocco avanz. asse Y Sens. Capacitivo in contatto con la lamiera
OR   Pul_Stop                      ** (gPlc0.2)Stop pushbutton
S    b_TipTouch                    ** (LsPlc47.7) TipTouch Attivo da MainFast

LDN  PRGSTOP_CN0                   ** (cn0.rc8.1)  Programma interrotto CN0
AND(
LD   Capacit_Anal_Mm		             ** (C103)Analogica Capacitivo in mm
LE   StandOff                      ** Valore distanza taglio in centesimi
)
ORN  PRGRUN_CN0                    ** M0.0 cn0.rc8.0  Programma in corso
R    b_TipTouch                    ** (LsPlc47.7) TipTouch Attivo da MainFast

***************************************
*   TIP TOUCH condition disable
***************************************
LD   %LSRPlcOp0.12                 ** Disable TIP TOUCH during piercing
AND  PRGRUN_CN0                    ** M0.0 cn0.rc8.0  Programma in corso
AND  (
LD   PiercingInRun                 ** (LsPlc70) Piercing in run
EQ   1
)
AND (
LD   Capacit_Anal_Mm		             ** (C103)Analogica Capacitivo in mm
LT   500                        ** < 5.00 mm
)
ST   appoggio3

CAL  TON_TIPTOUCH(IN=appoggio3,PT=500) ** Tip touch ritardato di 500 msec

LD   TON_TIPTOUCH.Q             ** Tip touch ritardato di 500 msec
ST   TipTouchDisable               ** (LsPlc71.0) TipTouchDisable (ritardato)

**************************************************
* Code for Hold retrace function
* - after [stop] button and retrace enabled
* - or after tip touch
**************************************************
LD   %FUNCBTN.1                            * [Stop]
AND  %LSRPlcOp1.16                 ** Enable retrace back after HOLD
OR   JogCommandTipTouch            ** (LsPlc47.0) Automatic jog command for tip touch
AND  %cn0.rc8.0                            * program in run
AND  iso_LsronCutting
S    appoggio4

LD   appoggio4
ANDN HW_PWM_CFG_FC                        ** Laser I/F board PWM_CFG register: FC
ST   appoggio

CAL  RTRIG_STOP(CLK:=appoggio)            * [Stop]

LD   RTRIG_STOP.Q
JMPCN  no_sample_dist

S    ch0stopusr                    ** Channel in stop from user request

LD   %ax21.ra25                           * Insterpolator distance
ST   dist1HoldPush                 ** Distance of the interpolator when Stop button is pushed

no_sample_dist:

LD  %cn0.rc8.1                            * channel in hold
AND (
LD  %ax27.ra3.0                           * axis X stop
AND %ax28.ra3.0                           * axis Y stop
)
JMPCN no_sample_dist2
LD   %ax21.ra25                           * Insterpolator distance
ST   dist2Hold                     ** Distance of the interpolator when axes are not moving any more
no_sample_dist2:

LD   dist2Hold                     ** Distance of the interpolator when axes are not moving any more
SUB  dist1HoldPush                 ** Distance of the interpolator when Stop button is pushed
ST   DeltaDist                     ** Delta distance for hold

CAL  FTRIG_RetrDone(CLK:=RetraceCommBack)          * (LsPlc47.11) Retrace command after hold)

LD   %FUNCBTN.0                           * [START]
OR   StartAftTipTouch              ** (LsPlc47.2) Start after tip touch
OR   RetrPlusReq                          ** (LsPlc47.9) Request of positive retrace, DO NOT REMOVE
OR   FTRIG_RetrDone.Q
ORN  %cn0.rc8.0                           * channel in run
OR   Pul_Reset                     ** (gPlc0.3)Reset pushbutton
R    ch0stopusr                    ** Channel in stop from user request
R    appoggio4

LD   ch0stopusr                    ** Channel in stop from user request
AND  (
LD   %ax21.ra25
GT   (
LD   dist1HoldPush                 ** Distance of the interpolator when Stop button is pushed
SUB  userdistance                  ** (LSRCostK54) User distance retrace
)
)
ST   appoggio

CAL  TON_RETRCOM(IN:=appoggio,PT:=200)

LD   TON_RETRCOM.Q
ST   RetraceCommBack                      * (LsPlc47.11) Retrace command after hold

**************************************************
* Regulation test
**************************************************
*******LD   %ax29.ra79
*******MUL  10
*******DIV  65536
*******MUL  1000
*******ST   %C127

**************************************************
* ECAT SAFETY
**************************************************
ECAT_SAFETY

**************************************************
* Pipe Welding
**************************************************
LD   %LSRPlcOp0.22                 ** Pipe Welding function enabling
JMPCN NoWeldingM

LD   WeldingFuncOn
ANDN WeldingNoRead
AND  I_I_WELDING_SENSOR
ST   appoggio

CAL  RTRIG_WELDING_COUNT(CLK:=appoggio)

LD   RTRIG_WELDING_COUNT.Q
JMPCN NoRead

LD   %ax34.ra4
ST   WeldingCfound

LD   WeldingSolderJointCoun
ADD  1
ST   WeldingSolderJointCoun

NoRead:
NoWeldingM:

**************************************************
* G0 Support to optimized lift
**************************************************
LD   IN_M700_M704
EQ   700
AND  %cn0.rc8.0
JMPCN RUNACTION

    LD   %gIso30                 * Optimized Lift - 19mm = hypotenuse_max
    SUB  19000
    SUB  %ax50.ra4
    ABS
    LT   1000                     * 0.5MM
    S    ParkUn71Sup_ISO
    S    ParkUn72Sup_ISO
    S    ParkUn73Sup_ISO
    S    ParkUn74Sup_ISO
    S    ParkUn75Sup_ISO
    S    ParkUn51Sup_ISO
    S    ParkUn52Sup_ISO
    S    ParkUn53Sup_ISO
    S    ParkUn54Sup_ISO

    LD   PreActbld
    SUB  %ax5.ra4
    ABS
    LT   5000                     * 5 degree
    ST   Appoggio
    CAL  R_TRIG_FOLLOW(CLK=Appoggio)

    LD   R_TRIG_FOLLOW.Q
    R    ParkUn71Sup_ISO
    R    ParkUn72Sup_ISO
    R    ParkUn73Sup_ISO
    R    ParkUn74Sup_ISO
    R    ParkUn75Sup_ISO
    R    ParkUn51Sup_ISO
    R    ParkUn52Sup_ISO
    R    ParkUn53Sup_ISO
    R    ParkUn54Sup_ISO
    S    M700_BLEND

    LD   R_TRIG_FOLLOW.Q
    JMPCN CLRSECFOLLOW
         LD 0
    	 ST SecFollow_51
    	 ST SecFollow_52
    	 ST SecFollow_53
    	 ST SecFollow_54
    	 ST SecFollow_71
    	 ST SecFollow_72
    	 ST SecFollow_73
    	 ST SecFollow_74
    	 ST SecFollow_75
    CLRSECFOLLOW:

RUNACTION:

********************************************************
* Pgm Loading Finished (2.5ms TP right after finishing)
* ---> Add 7.5ms to be 10ms
********************************************************
LD    %PlcOp0.29
ST    EnBvlConerOptim

CAL   F_TRIG_PGMSEND(CLK=%ui16.30)
CAL   TP_PGMSEND(IN=F_TRIG_PGMSEND.Q,PT=3000)
LD    TP_PGMSEND.Q
AND   EnBvlConerOptim
ST    CornerChangeCmd
ST    CorOptNoStart

END_FUNCTION

(* ---- MConfig.plc ---- *)
*******************************************************************************
*   MCONFIG.PLC
*   ESAutomotion
*   LASER machine
*******************************************************************************
#funcdec "FBAux.plc"
#funcdec "res_ipg.plc"
#funcdec "LsrGest.plc"
#funcdec "CAP_Prec.plc"
#funcdec "FocProco.plc"
#funcdec "Foc_Prec.plc"
#funcdec "nLight.plc"
#funcdec "CAP_EMP.plc"

VAR
#include "Cnc.inc"
#include "Iof.inc"
END_VAR

VAR_IN_OUT
#include "mem.inc"
END_VAR

#include "Iol.inc"
#include "res_ipg.inc"
**#include "LsrGest.inc"
#include "Cap_Prec.inc"
#include "foc_prec.inc"

VAR
CAP_PROCON_0:           CAP_PREC;
CAP_EMP_0:              CAP_EMP;
Focal_Precitec:         FOC_PRECITEC;
IPG_0:                  IPG;
NLIGHT0:                NLIGHT;
LSRGEST_0:              LSRGST;
LASER_SHOOT_0:          LASER_SHOOT;
appoggio:               BOOL;
Aux_Allarme:            BOOL;
Hold_Emission_ON:       BOOL;
TOF_Restart_Laser:      TOF;        * Ritardo accensione Laser dopo OVR=0 o NC_STOP
F_TRIG_HOLD:            F_TRIG;
TP_HOLD:                TP;         * Tempo inibiz.Uscita Emissione dopo Hold (Per stabil.Pressioni Gas)
TON1:                   TON;        * Attesa per emissione allarme
LaserSim:               BOOL;
TOF_REF_HEAD:           TOF;
temp:                   DWORD;
END_VAR

*******************************************************************************
*   MACHINE CONFIGURATION
*******************************************************************************
FUNCTION MACHINE_CONFIG

***************************************
*   PROCON CAPACITIVE
***************************************
PATH %Capacitive[0]

LD   %config_machine26
EQ   0
OR(
LD   %config_machine26
EQ   4
)
JMPCN no_prec_cap

LD   Memo_Emission_ON_da_Funz_M    ** M107.25 Memoria Emission ON da Funzione M
ST   CAP_PROCON_0.xEmission

CAL  CAP_PROCON_0

LD   CAP_PROCON_0.yMsg.0
ST   %PLCmsg4.0                 * PLC Msg 128 Calibrazione in corso

LD   CAP_PROCON_0.yMsg.1
ST   %PLCmsg7.0

LD   CAP_PROCON_0.yErr.0
ST   %PLCerr5.4                 * PLC Err 164 Tip touch (A11=1, A14=0, A15=0 in normal operation)

LD   CAP_PROCON_0.yErr.1
ST   %PLCerr5.5                 * PLC Err 165 Body touch (A11=1, A14=1, A15=0 in normal operation)

LD   CAP_PROCON_0.yErr.2
ST   %PLCerr5.6                 * PLC Err 166 Nozzle lost (A11=1, A14=0, A15=1 in normal operation)

LD   CAP_PROCON_0.yErr.3
ST   %PLCerr5.7                 * PLC Err 167 Tempo massimo calibrazione sensore capacitivo

LD   CAP_PROCON_0.yErr.4
ST   %PLCerr5.8                 * PLC Err 168 Cable cut da capacitivo

LD   CAP_PROCON_0.yErr.5
ST   %PLCmsg7.13                * Check FAR e/o CAPACITIVE

LD   CAP_PROCON_0.yExeCalib
ST   ExeCalibraz                   ** (LsPlc11.0) Richiesta esecuzione Calibrazione

LD   CAP_PROCON_0.yTipTouch
ST   TipTouchNotFiltered

***************************************
*** Signal from inputs managed in ISO fixed cycle
LD   I_FAR_A10                     ** Far away
ST   ISO_I_FAR_A10                 ** (C31.0) FAR input (used in ISO, into calibration fun)
LD   I_TIP_BODY_TOUCH_A11          ** Tip\Body Touch or Nozzle_Lost (TIP TOUCH:A11=1,A14=0,A15=0)
ST   ISO_I_TIP_BODY_TOUCH_A11      ** (C31.1) Tip-Body Touch o Nozzle_Lost (used in ISO, into calibration fun)
LD   I_READY_A13                   ** Ready
ST   ISO_I_READY_A13               ** (C31.2) READY (used in ISO, into calibration fun)
LD   I_NOZZLE_LOST_A15             ** Nozzle Lost/Pos reached (NOZZLE LOST:A11=1,A14=0,A15=1)
ST   ISO_I_NOZZLE_LOST_A15         ** (C31.3) POS reached (used in ISO, into calibration fun)

*** Command to manage output from ISO fixed cycle
LD   ISO_O_CALIB_REQ               ** (C30.7) Calibration request from ISO
AND  ExeCalibraz                   ** (LsPlc11.0) Richiesta esecuzione Calibrazione
ST   O_CALIBRA_REQ_A3              ** Calibration request

LD   ISO_O_CALIB_STROBE            ** (C30.8) Calibration strobe from ISO
AND  ExeCalibraz                   ** (LsPlc11.0) Richiesta esecuzione Calibrazione
ST   O_STROBE_A7                   ** Strobe

no_prec_cap:

***************************************
*   EMPOWER CAPACITIVE
***************************************
LD   %config_machine26
EQ   3
JMPCN no_empower_cap

LD   Memo_Emission_ON_da_Funz_M    ** M107.25 Memoria Emission ON da Funzione M
ST   CAP_EMP_0.xEmission

LD   IA_Emower_cap
ST   CAP_EMP_0.xEmp_sensor

CAL  CAP_EMP_0

LD   CAP_EMP_0.yMsg.0
ST   %PLCmsg4.0                 * PLC Msg 128 Calibrazione in corso

LD   CAP_EMP_0.yErr.0
ST   %PLCerr5.4                 * PLC Err 164 Tip touch (A11=1, A14=0, A15=0 in normal operation)

LD   CAP_EMP_0.yErr.3
ST   %PLCerr5.7                 * PLC Err 167 Tempo massimo calibrazione sensore capacitivo

LD   CAP_EMP_0.yErr.4
ST   %PLCerr5.8                 * PLC Err 168 Cable cut da capacitivo

LD   CAP_EMP_0.yExeCalib
ST   ExeCalibraz                   ** (LsPlc11.0) Richiesta esecuzione Calibrazione

LD   CAP_EMP_0.yTipTouch
ST   TipTouchNotFiltered

LD   CAP_EMP_0.yFar
ST   %EmConfig.Far_signal.0

***************************************
*** Signal from inputs managed in ISO fixed cycle

LD   CAP_EMP_0.yTipTouch
ST   ISO_I_TIP_BODY_TOUCH_A11      ** (C31.1) Tip-Body Touch o Nozzle_Lost (used in ISO, into calibration fun)

no_empower_cap:

***************************************
*   PROCON FOCAL
***************************************
LD   %config_machine25
EQ   4
JMPCN no_procon
     PROCON_FOCAL    * not used
no_procon:

***************************************
*   PRECITEC FOCAL
***************************************
LD   %config_machine25
EQ   0
JMPCN no_prec

PATH %Head_Laser[0]

LD   %TabLsr0.L_CutFocal             ** Valore focale passato da tabelle
ST   temp

***************************************
*   Focal=funz(angle)
*   #CDL
***************************************
LD   PRGRUN_CN0
ANDN PRGSTOP_CN0
AND (
LD   %uvHeads0.uvhCommand1
EQ   4                              * Cutting phase
)
AND  %LSRPlcOp0.3
JMPCN no_corr_focal

LD   temp
ADD (
LD   temp
MULDIV(M=%TsCutDataLinear.CDL_Focal,D=100000) * 100 %
)
ST   temp

no_corr_focal:
*
***************************************

LD   temp
ST   Focal_Precitec.xCutFoc

LD   Val_Focale_ACT                 ** Valore Focale da\a GUI
ST   Focal_Precitec.xVal_Focale_ACT

LD   %config_machine30
ST   Focal_Precitec.xAnRes

LD   Focal_Type
ST   Focal_Precitec.xFocal_Type

CAL  Focal_Precitec

LD   Focal_Precitec.yFocAn
ST   OA_FOCALE

LD   Focal_Precitec.yPrec_Pos_Run
ST   Prec_Pos_Run                  ** Focal positioning in run (Used Piercing ISO)

LD   Focal_Precitec.yError.0       * Precitec: reference error
S    %PLCerr5.1

LD   Focal_Precitec.yError.1       * Precitec: reference timeout
S    %PLCerr5.3

LD   Focal_Precitec.yError.2       * General Precitec Error
S    %PLCerr7.7

LD   Focal_Precitec.yError.3       * Precitec: lens/prot. not present
S    %PLCerr5.0

LD   Focal_Precitec.yError.4       * Precitec: automatic error
S    %PLCerr5.2

LD   Focal_Precitec.yMsg.0         * Precitec: lens not present (SW1)
S    %PLCmsg5.0

LD   Focal_Precitec.yMsg.1         * Precitec: protective lens not present (SW4)
S    %PLCmsg5.1

LD   Focal_Precitec.yMsg.2         * Precitec: reference completed
S    %PLCmsg5.2

no_prec:

LD   RESET_ALLARMI
R    %PLCerr5.0
R    %PLCerr5.1
R    %PLCerr5.2
R    %PLCerr5.3
R    %PLCerr7.7
R    %PLCmsg5.0
R    %PLCmsg5.1
R    %PLCmsg5.2

***************************************
*   IPG RESONATOR
***************************************
PATH %LsrGest[0]

LD   %ParOptions.0
ST   LaserSim

LD   %TabLsr0.L_CutPower
ST   LSRGEST_0.xPower

LD   %TabLsr0.L_CutDuty
ST   LSRGEST_0.xDuty

LD   %TabLsr0.L_CutFreq
ST   LSRGEST_0.xFreq

CAL  LSRGEST_0

***LD   LSRGEST_0.yEmission
***ST   Memo_Emission_ON_da_Funz_M    ** M107.25 Memoria Emission ON da Funzione M

* If shoot is managed in lsrgest, FC out output
LD   LSRGEST_0.yEmission
ST   LaserOn                       ** (LsPlc1.25) Per GUI  LaserOn
***************************************

PATH %Resonator[0]

LD   0              * YLS
ST   IPG_0.xType

LD   LaserSim
OR (
LD   CMD_RESONATOR_OFF
EQ   1
)
ST   IPG_0.xSIM

LD   Pul_Reset                     ** (gPlc0.3)Reset pushbutton
ST   IPG_0.xReset

LD   EMER_GEN
ST   IPG_0.xEmer

LD   Ordine_Moto_X1                ** M71.0 Ordine di moto asse X1
OR   Ordine_Moto_Y1                ** M71.8 Ordine di moto asse Y1
AND  %PLCmsg0.19    ** Feedrate a ZERO
OR   SPURGOrun                     ** M107.2 Gas purge in progress
OR   PRGSTOP_CN0                   ** (cn0.rc8.1)  Programma interrotto CN0
ST   Hold_Emission_ON   ** Condizioni per Hold Emission_ON Laser

CAL  TOF_Restart_Laser(IN=Hold_Emission_ON,PT=500) ** Ritardo accensione Laser dopo OVR=0 o NC_STOP
LD   TOF_Restart_Laser.Q            ** Ritardo accensione Laser dopo OVR=0 o NC_STOP
***OR   TP_HOLD.Q                       * Tempo inibiz.Uscita Emissione dopo Hold (Per stabil.Pressioni Gas)
ANDN (
LD   RetrPlusReq                   ** (LsPlc47.9) Request of positive retrace
OR   RetrMinusReq                  ** (LsPlc47.10) Request of negative retrace
)
ST  BL_AV_ASSI_X_OVR               ** M74.8 Blocco avanzamento assi dopo Override=0 o NC_STOP

CAL F_TRIG_HOLD(CLK=M_HOLD)        ** (gPlc19.0)Mem. Richiesta Hold

LD   F_TRIG_HOLD.Q
AND  PRGRUN_CN0                    ** M0.0 cn0.rc8.0  Programma in corso
ST   appoggio
CAL  TP_HOLD(IN=appoggio,PT=3000)  ** Tempo inibiz.Uscita Emissione dopo Hold (Per stabil.Pressioni Gas)

LD   Memo_Emission_ON_da_Funz_M    ** M107.25 Memoria Emission ON da Funzione M
ANDN Hold_Emission_ON              ** Condizioni per Hold Emission_ON Laser
ANDN M_HOLD                        ** (gPlc19.0)Mem. Richiesta Hold
ANDN %PLCerr5.4                    **PLC Err 164 Tip touch (A11=1, A14=0, A15=0 in normal operation)
ANDN TP_HOLD.Q                     * Tempo inibiz.Uscita Emissione dopo Hold (Per stabil.Pressioni Gas)
ANDN DryRunOption                  ** Macchina in modo Dry Run
ANDN IPG_0.xSIM
ST   IPG_0.xEmission

CAL  IPG_0

LD   IPG_0.yError.0
S    %PLCerr5.19                    *IPG laser error (B4)

LD   IPG_0.yError.1
S    %PLCerr5.18                    *IPG laser not ready (A2 without B1)

LD   IPG_0.yError.2
S    %PLCerr5.16                    *IPG laser not assigned (A1 without B7)

LD   IPG_0.yError.3
S    %PLCerr5.17                    *IPG laser not ready (C1 without B8)

LD   IPG_0.yError.4
S    %PLCerr5.20                    *IPG Timeout feedback emission ON

*LD   IPG_0.yState
*ST   LaserOn                       ** (LsPlc1.25) Per GUI  LaserOn

* Allarme : Comandata emissione laser con valvole chiuse
LD   IPG_0.yState
ANDN O_O_EV_OR_ALLGAS              ** M90.15 Elettrovalvola apertura di almeno un gas
ANDN %PlcOp0.2                     ** DryRun
ST   Aux_Allarme

CAL  TON1(IN=Aux_Allarme,PT=500)   ** Attesa per emissione allarme

LD   TON1.Q
S    %PLCerr5.21                    *IPG Comandata emissione laser con valvole chiuse

LD   RESET_ALLARMI                 ** M100.4  Cancellazione allarmi attiva
OR   LaserSim
R    %PLCerr5.16                    *IPG laser not assigned (A1 without B7)
R    %PLCerr5.17                    *IPG laser not ready (C1 without B8)
R    %PLCerr5.18                    *IPG laser not ready (A2 without B1)
R    %PLCerr5.19                    *IPG laser error (B4)
R    %PLCerr5.20                    *IPG Timeout feedback emission ON
R    %PLCerr5.21                    *IPG Comandata emissione laser con valvole chiuse

********************************************************************************
* nLight
LD   %config_machine28
EQ   5
JMPCN NLIGHTSEL                     *nlight
PATH %Resonator[1]

LDN  I_I_EMERGENZA
ST   NLIGHT0.xEmer

CAL  NLIGHT0
NLIGHTSEL:

***************************************
*   LASER SHOOT
***************************************
PATH %FocalPwm[0]

PATH %LsrGest[0]

CAL  LASER_SHOOT_0

LD   LASER_SHOOT_0.yShootOn
ST   %LaserShootOn

LD   %TstP15
EQ   0
ST   UnlockLaserComm

END_FUNCTION

(* ---- OnOfMac.plc ---- *)
*******************************************************************************
*   ONOFFMAC.PLC
*   ESAutomotion
*   LASER machine
*******************************************************************************
VAR
#include "Cnc.inc"
#include "RemContr.inc"

FPN_MACCH_ON:       TRIG;       * Fronte salita\discesa macchina ON
TON_ALLARM:     	TON;        * TON salita allarme
RTRIG_REM_DRY:      R_TRIG;

END_VAR

VAR_IN_OUT
#include "mem.inc"
END_VAR

#include "Iol.inc"

*******************************************************************************
* Gestione Accensione\Spegnimento macchina e RESET
*******************************************************************************
FUNCTION Macch_Reset

*******************************************************************************
*   EMERGENZA MACCHINA DA  CN, PLC, Comando Sbloccaggio Protezioni Macchina
*******************************************************************************
LDN  O_O_CNC_OK                    ** CNC OK
***(TODO)OR   EMERG_DA_SBL_PROTEZ
ST   EMERGENZA_PLC_CN              ** M100.0  Emergenza da PLC o da CN

*******************************************************************************
*   Macchina OK
*******************************************************************************
LDN  I_I_EMERGENZA                 ** Machine OK (no EMERG.)
ST   MACCHINA_OK                   ** M100.1  Macchina OK

*******************************************************************************
*   Ciclo di Reference GENERALE in corso
*******************************************************************************
LD   REF_RUN                       ** M0.12 Taratura in corso
ANDN PLC_SEL_SINGREF               ** ui16.28 Selezione REF singolo
ST   GEN_REF_RUN                   ** M100.16 Ciclo di Reference GENERALE in corso

*******************************************************************************
*   Macchina in MANUALE
*******************************************************************************
LD   ch3_in_jog                    ** channel 3 in jog
ST   MACCH_IN_MANUALE              ** M100.24 SELEZIONE MACCHINA IN MANUALE

*******************************************************************************
*   Macchina in AUTOMATICO
*******************************************************************************
LD   ch3_in_aut                    ** channel 3 in aut
ST   MACCH_IN_AUTO                 ** M100.25 SELEZIONE MACCHINA IN AUTOMATICO

*******************************************************************************
*   Macchina in SIMULAZIONE
*******************************************************************************
CAL  RTRIG_REM_DRY(CLK:=RemContrDryRun)    * Xhc_Puls.8  Select Dry Run

LD   RTRIG_REM_DRY.Q
AND  DryRunOption                   ** Macchina in modo Dry Run
JMPCN no_dry_run
LD   0
ST   DryRunOption                   ** Macchina in modo Dry Run
JMP no_dry
no_dry_run:

LD   RTRIG_REM_DRY.Q
ANDN DryRunOption                   ** Macchina in modo Dry Run
JMPCN yes_dry_run
LD   1
ST   DryRunOption                   ** Macchina in modo Dry Run
yes_dry_run:
no_dry:

LD      %PlcOp0.2                ** Macchina in modo Dry Run
ST      MACCH_IN_SIM	              ** M100.28 MACCHINA IN SIMULAZIONE

*******************************************************************************
*  SICUREZZE RIPRISTINATE (ON MACCHINA)
*******************************************************************************
CAL  FPN_MACCH_ON(CLK:=MACCHINA_OK) ** Fronte salita\discesa macchina ON

LD   FPN_MACCH_ON.Q
AND  MACCHINA_OK                   ** M100.1  Macchina OK
ST   FP_MACCHINA_ON                ** M100.8  Fronte di salita Macchina ON

LD   FPN_MACCH_ON.Q
ANDN MACCHINA_OK                   ** M100.1  Macchina OK
ST   FN_MACCHINA_ON                ** M100.7  Fronte di discesa Macchina ON

*******************************************************************************
*  RESET DA PULSANTE O AD ACCENSIONE MACCHINA
*******************************************************************************
LD   Pul_Reset                     ** (gPlc0.3)Reset pushbutton
OR   FP_MACCHINA_ON                ** M100.8  Fronte di salita Macchina ON
ST   RESET_MACCHINA                ** M100.2  Reset macchina

******************************************************
*  CANCELLAZIONE ALLARMI E MESSAGGI
******************************************************
LD   ON_ONE_SCAN                  ** PLCFLAGS.8  Flag on alla prima scansione PLC
OR   RESET_MACCHINA                ** M100.2  Reset macchina
ST   RESET_ALLARMI                 ** M100.4  Cancellazione allarmi attiva

******************************************************
*  AUTO JOG MODE
******************************************************
LD   RemContrYPlus
OR   RemContrCMinus
OR   RemContrUPlus
OR   RemContrUMinus
OR   RemContrCPlus
OR   RemContrZPlus
OR   RemContrXMinus
OR   RemContrXPlus
OR   RemContrYMinus
OR   RemContrZMinus
OR   Gui_btn_CW
OR   Gui_btn_CCW
OR   Gui_Pul_X_M
OR   Gui_Pul_X_P
OR   Gui_Pul_X1_M
OR   Gui_Pul_X1_P
OR   Rem_Combination
ANDN %cn0.rc8.0
ST   ContrJogFromBtn

******************************************************
*   ALLARME ATTIVO
******************************************************
LD  %PLCerr0
GT  0
OR(
LD  %PLCerr1
GT  0
)
OR(
LD  %PLCerr2
GT  0
)
OR (
LD  %PLCerr3
GT  0
)
OR (
LD  %PLCerr4
GT  0
)
OR (
LD  %PLCerr5
GT  0
)
OR (
LD  %PLCerr6
GT  0
)
ST   ALARM_ACT                     ** M100.3  Allarme attivo

END_FUNCTION
